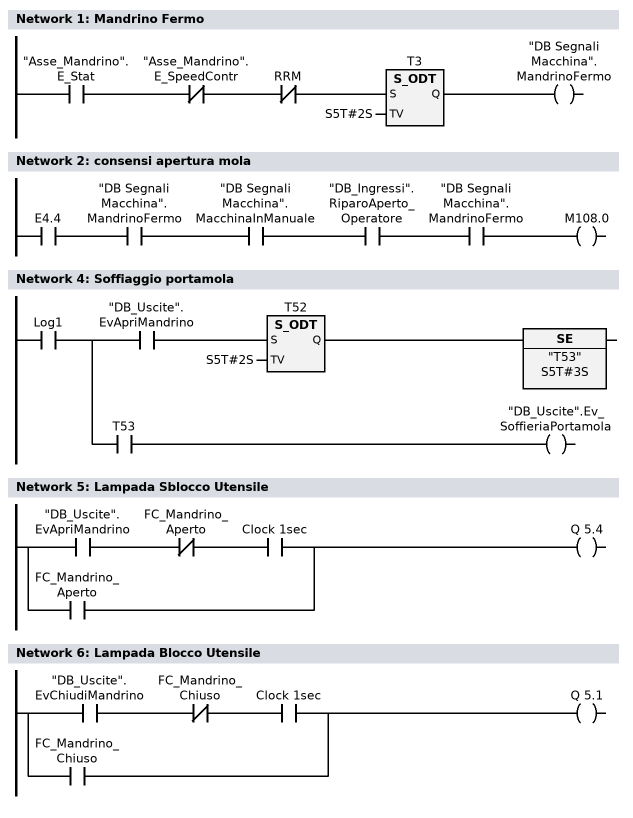
NETWORK
TITLE = Mandrino Fermo
      A     "Asse_Mandrino".E_Stat;
      AN    "Asse_Mandrino".E_SpeedContr;
      AN    "RRM";
      L     S5T#2S;
      SD    "T3";
      NOP   0;
      NOP   0;
      NOP   0;
      A     "T3";
      =     "DB Segnali Macchina".MandrinoFermo;
NETWORK
TITLE = consensi apertura mola
      A     "E4.4";
      A     "DB Segnali Macchina".MandrinoFermo;
      A     "DB Segnali Macchina".MacchinaInManuale;
      A     "DB_Ingressi".RiparoAperto_Operatore;
      A     "DB Segnali Macchina".MandrinoFermo;
      =     "M108.0";
NETWORK
TITLE = Blocco - Sblocco Mandrino
      A(;
      A(;
      A     "Pulsantiera.ChiudiMand";
      L     S5T#2S;
      SD    "T54";
      NOP   0;
      NOP   0;
      NOP   0;
      A     "T54";
      );
      A     "DB Segnali Macchina".MacchinaInManuale;
      A     "DB Segnali Macchina".MandrinoFermo;
      R     "DB_Uscite".EvApriMandrino;
      A(;
      A     "Pulsantiera.ApriMand";
      L     S5T#2S;
      SD    "T55";
      NOP   0;
      NOP   0;
      NOP   0;
      A     "T55";
      );
      A     "M108.0";
      S     "DB_Uscite".EvApriMandrino;
      A     "DB_Uscite".EvApriMandrino;
      );
      NOT;
      =     "DB_Uscite".EvChiudiMandrino;
NETWORK
TITLE = Soffiaggio portamola
      A     "Log1";
      =     L 0.0;
      A     L 0.0;
      A     "DB_Uscite".EvApriMandrino;
      L     S5T#2S;
      SD    "T52";
      NOP   0;
      NOP   0;
      NOP   0;
      A     "T52";
      L     S5T#3S;
      SE    "T53";
      A     L 0.0;
      A     "T53";
      =     "DB_Uscite".Ev_SoffieriaPortamola;
NETWORK
TITLE = Lampada Sblocco Utensile
      A     "DB_Uscite".EvApriMandrino;
      AN    "FC_Mandrino_Aperto";
      A     "Clock 1sec";
      O     "FC_Mandrino_Aperto";
      =     Q 5.4;
NETWORK
TITLE = Lampada Blocco Utensile
      A     "DB_Uscite".EvChiudiMandrino;
      AN    "FC_Mandrino_Chiuso";
      A     "Clock 1sec";
      O     "FC_Mandrino_Chiuso";
      =     Q 5.1;
END_FUNCTION

FUNCTION "FC Refrigerante" : VOID	// FC 106
TITLE = Gestione Refrigerante
AUTHOR : Asamec
VERSION : 0.1
BEGIN
NETWORK
TITLE = Refrigerante 1
      A(;
      A(;
      A     "Pulsantiera.AccendiOlio1";
      FP    "M10.0";
      =     "M93.2";
      A     "M93.2";
      AN    "DB_Ingressi".RiparoAperto_Operatore;
      A     "DB_Ingressi".RiparoChiuso_Robot;
      AN    "DB_Ingressi".Sel_MAN_AUTO;
      O     "M07";
      O;
      A     "M08";
      A(;
      L     "Chan1".T1;
      L     1;
      ==I;
      );
      );
      S     "M33.0";
      A(;
      O     "Pulsantiera.Reset";
      O;
      A     "Pulsantiera.SpegniOlio";
      AN    "DB_Ingressi".Sel_MAN_AUTO;
      ON    "DB Segnali Macchina".MacchinaAccesa;
      O     "M09";
      O;
      A     "M08";
      A(;
      L     "Chan1".T1;
      L     2;
      ==I;
      );
      A     "DB_Ingressi".Sel_MAN_AUTO;
      );
      R     "M33.0";
      A     "M33.0";
      );
      AN    "DB_Ingressi".RiparoAperto_Operatore;
      A     "DB_Ingressi".RiparoChiuso_Robot;
      AN    "M92.3";
      AN    "DB Allarmi".Canale1.Feed_And_Read_Disable.A510119;
      AN    "DB Allarmi".Canale1.Feed_And_Read_Disable.A510120;
      AN    "DB Allarmi".Canale1.Feed_Disable.A510004;
      AN    "DB Allarmi".Canale1.Feed_And_Read_Disable.A510117;
      =     "DB_Uscite".Olio1;
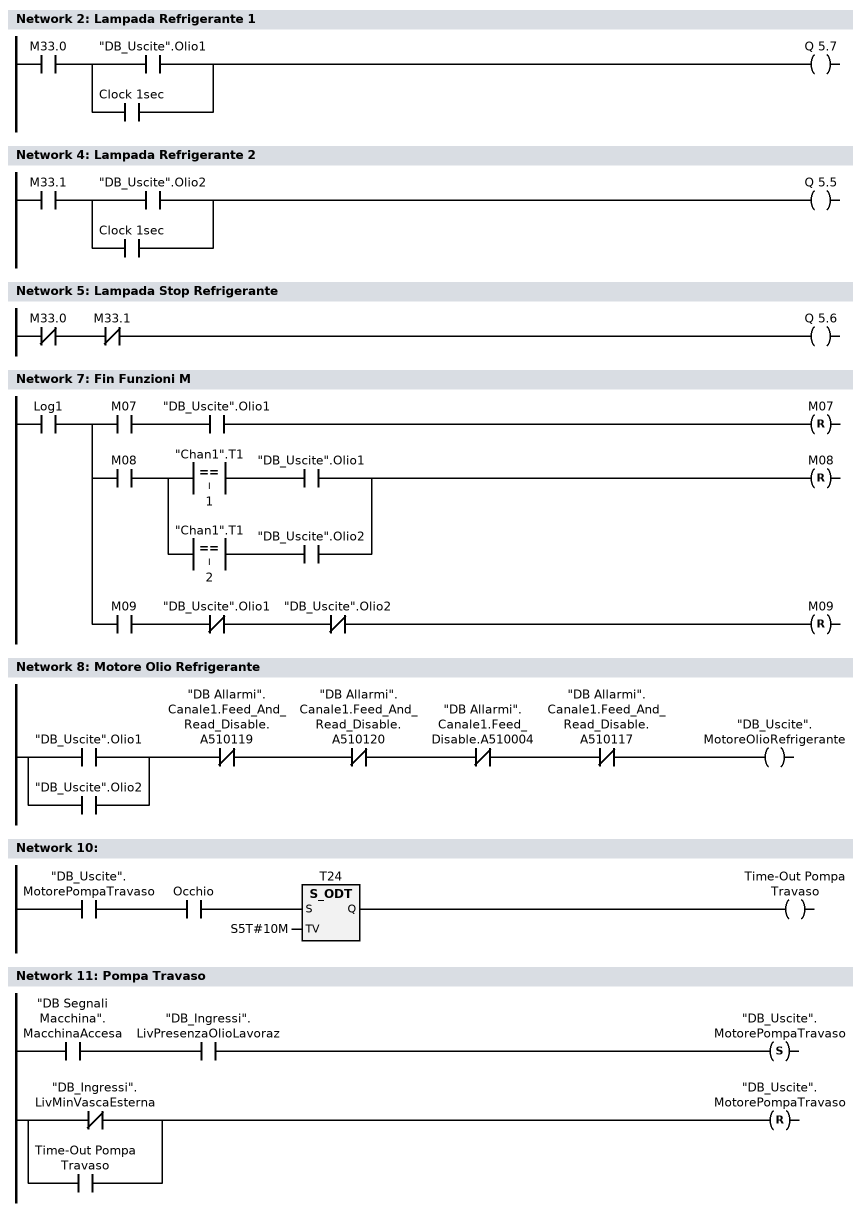
NETWORK
TITLE = Lampada Refrigerante 1
      A     "M33.0";
      A(;
      O     "DB_Uscite".Olio1;
      O     "Clock 1sec";
      );
      =     Q 5.7;
NETWORK
TITLE = Refrigerante 2
      A(;
      A(;
      A     "Pulsantiera.AccendiOlio2";
      FP    "M10.1";
      =     "M93.3";
      A     "M93.3";
      AN    "DB_Ingressi".RiparoAperto_Operatore;
      A     "DB_Ingressi".RiparoChiuso_Robot;
      AN    "DB_Ingressi".Sel_MAN_AUTO;
      O;
      A     "M08";
      A(;
      L     "Chan1".T1;
      L     2;
      ==I;
      );
      );
      S     "M33.1";
      A(;
      O     "Pulsantiera.Reset";
      O;
      A     "Pulsantiera.SpegniOlio";
      AN    "DB_Ingressi".Sel_MAN_AUTO;
      ON    "DB Segnali Macchina".MacchinaAccesa;
      O     "M09";
      O;
      A(;
      L     "Chan1".T1;
      L     1;
      ==I;
      );
      A     "DB_Ingressi".Sel_MAN_AUTO;
      );
      R     "M33.1";
      A     "M33.1";
      );
      AN    "DB_Ingressi".RiparoAperto_Operatore;
      A     "DB_Ingressi".RiparoChiuso_Robot;
      AN    "M92.3";
      AN    "DB Allarmi".Canale1.Feed_And_Read_Disable.A510119;
      AN    "DB Allarmi".Canale1.Feed_And_Read_Disable.A510120;
      AN    "DB Allarmi".Canale1.Feed_Disable.A510004;
      AN    "DB Allarmi".Canale1.Feed_And_Read_Disable.A510117;
      =     "DB_Uscite".Olio2;
NETWORK
TITLE = Lampada Refrigerante 2
      A     "M33.1";
      A(;
      O     "DB_Uscite".Olio2;
      O     "Clock 1sec";
      );
      =     Q 5.5;
NETWORK
TITLE = Lampada Stop Refrigerante
      AN    "M33.0";
      AN    "M33.1";
      =     Q 5.6;
NETWORK
TITLE = Sospendi refrigerante in automatico
      A     "Pulsantiera.SpegniOlio";
      A     "DB_Ingressi".Sel_MAN_AUTO;
      FP    "M93.1";
      X     "M92.3";
      =     "M92.3";
      A     "M07";
      O     "M08";
      ON    "DB_Ingressi".Sel_MAN_AUTO;
      R     "M92.3";
NETWORK
TITLE = Fin Funzioni M
      A     "Log1";
      =     L 0.0;
      A     L 0.0;
      A     "M07";
      A     "DB_Uscite".Olio1;
      R     "M07";
      A     L 0.0;
      A     "M08";
      A(;
      A(;
      L     "Chan1".T1;
      L     1;
      ==I;
      );
      A     "DB_Uscite".Olio1;
      O;
      A(;
      L     "Chan1".T1;
      L     2;
      ==I;
      );
      A     "DB_Uscite".Olio2;
      );
      R     "M08";
      A     L 0.0;
      A     "M09";
      AN    "DB_Uscite".Olio1;
      AN    "DB_Uscite".Olio2;
      R     "M09";
NETWORK
TITLE = Motore Olio Refrigerante
      A(;
      O     "DB_Uscite".Olio1;
      O     "DB_Uscite".Olio2;
      );
      AN    "DB Allarmi".Canale1.Feed_And_Read_Disable.A510119;
      AN    "DB Allarmi".Canale1.Feed_And_Read_Disable.A510120;
      AN    "DB Allarmi".Canale1.Feed_Disable.A510004;
      AN    "DB Allarmi".Canale1.Feed_And_Read_Disable.A510117;
      =     "DB_Uscite".MotoreOlioRefrigerante;
NETWORK
TITLE = Gestione Livelli
NETWORK
TITLE =
      A     "DB_Uscite".MotorePompaTravaso;
      A     "Occhio";
      L     S5T#10M;
      SD    "T24";
      NOP   0;
      NOP   0;
      NOP   0;
      A     "T24";
      =     "Time-Out Pompa Travaso";
NETWORK
TITLE = Pompa Travaso
      A     "DB Segnali Macchina".MacchinaAccesa;
      A     "DB_Ingressi".LivPresenzaOlioLavoraz;
      S     "DB_Uscite".MotorePompaTravaso;
      A(;
      ON    "DB_Ingressi".LivMinVascaEsterna;
      O     "Time-Out Pompa Travaso";
      );
      R     "DB_Uscite".MotorePompaTravaso;
      NOP   0;
NETWORK
TITLE =
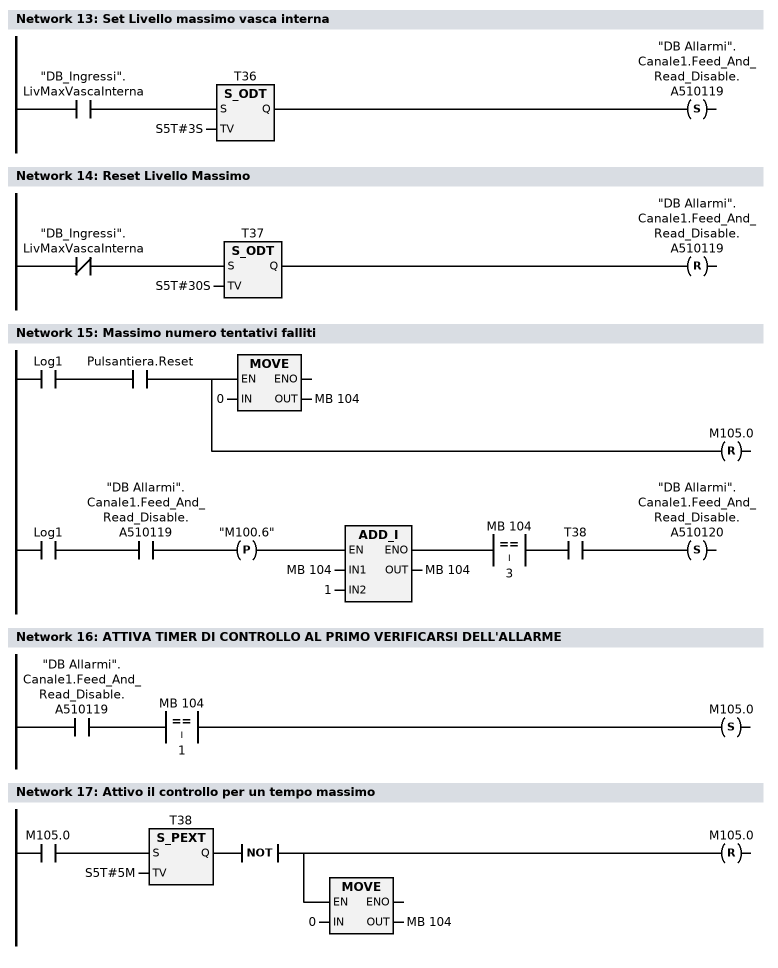
NETWORK
TITLE = Set Livello massimo vasca interna
      A     "DB_Ingressi".LivMaxVascaInterna;
      L     S5T#3S;
      SD    "T36";
      NOP   0;
      NOP   0;
      NOP   0;
      A     "T36";
      S     "DB Allarmi".Canale1.Feed_And_Read_Disable.A510119;
NETWORK
TITLE = Reset Livello Massimo
      AN    "DB_Ingressi".LivMaxVascaInterna;
      L     S5T#30S;
      SD    "T37";
      NOP   0;
      NOP   0;
      NOP   0;
      A     "T37";
      R     "DB Allarmi".Canale1.Feed_And_Read_Disable.A510119;
NETWORK
TITLE = Massimo numero tentativi falliti
      A     "Log1";
      =     L 0.0;
      A(;
      A     L 0.0;
      A     "DB Allarmi".Canale1.Feed_And_Read_Disable.A510119;
      FP    "M100.6";
      JNB   _001;
      L     MB 104;
      L     1;
      +I;
      T     MB 104;
      AN    OV;
      SAVE;
      CLR;
_001: A     BR;
      );
      A(;
      L     MB 104;
      L     3;
      ==I;
      );
      A     "T38";
      S     "DB Allarmi".Canale1.Feed_And_Read_Disable.A510120;
      A     L 0.0;
      A     "Pulsantiera.Reset";
      =     L 0.1;
      A     L 0.1;
      JNB   _002;
      L     0;
      T     MB 104;
_002: NOP   0;
      A     L 0.1;
      BLD   102;
      R     "M105.0";
NETWORK
TITLE = ATTIVA TIMER DI CONTROLLO AL PRIMO VERIFICARSI DELL'ALLARME
      A     "DB Allarmi".Canale1.Feed_And_Read_Disable.A510119;
      A(;
      L     MB 104;
      L     1;
      ==I;
      );
      S     "M105.0";
NETWORK
TITLE = Attivo il controllo per un tempo massimo
      A(;
      A     "M105.0";
      L     S5T#5M;
      SE    "T38";
      NOP   0;
      NOP   0;
      NOP   0;
      A     "T38";
      );
      NOT;
      =     L 0.0;
      A     L 0.0;
      BLD   102;
      R     "M105.0";
      A     L 0.0;
      JNB   _003;
      L     0;
      T     MB 104;
_003: NOP   0;
END_FUNCTION

FUNCTION "FC Assi" : VOID	// FC 107
VERSION : 0.1
BEGIN
NETWORK
TITLE =
NETWORK
TITLE = Abilita potenza OFF1 ( ex 48 - 112)
      A     "NC".E_DrivesInCylOp;
      A     "DB_Ingressi".AlimentatorePronto;
      A     "DB_Ingressi".PotenzaDriveInserita;
      S     "DB_Uscite".CdoOFF1;
      AN    "DB_Ingressi".PotenzaDriveInserita;
      R     "DB_Uscite".CdoOFF1;
NETWORK
TITLE = Abilita impulsi OFF3 ( ex 663 )
      A     "DB_Uscite".CdoOFF1;
      A     "DB_Ingressi".AusiliariInseriti;
//      U     "DB_Ingressi".PotenzaDriveInserita
      =     "DB_Uscite".CdoOFF3;
NETWORK
TITLE = Abilitazione assi
      A     "DB_Uscite".CdoOFF3;
//      U     "DB_Ingressi".ModuloARattivo
      =     "ConsensoRegolatore_X";
      =     "AbilitaImpulsi_X";
//-
      =     "ConsensoRegolatore_Y";
      =     "AbilitaImpulsi_Y";
//-
      =     "ConsensoRegolatore_Z";
      =     "AbilitaImpulsi_Z";
//-
NETWORK
TITLE = Abilitazione assi a e b (stop se fermi)
      A     "DB_Uscite".CdoOFF3;
      AN    "DB_Uscite".EV_ApriPortaPezzo;
      =     "M90.0";
      A     "Asse A in Direzione -";
      O     "Asse A in Direzione +";
      O     "BAG".E_AUTO;
      ON    "Chan1".E_ChanReset;
      A     "DB_Ingressi".AusiliariInseriti;
      S     "M90.1";
      R     "DB_Uscite".BloccoAsseA;
      A     "M90.0";
      A     "M90.1";
      AN    "DB_Ingressi".PressTavolaOrizzontale;
      AN    "DB_Uscite".EV_ApriPortaPezzo;
      L     S5T#200MS;
      SD    T 41;
//-
      A     T 41;
      S     "ConsensoRegolatore_A";
      S     "AbilitaImpulsi_A";
//-
      AN    "Asse A in Direzione -";
      AN    "Asse A in Direzione +";
      A     "Asse A Fermo";
      AN    "BAG".E_AUTO;
      A     "Chan1".E_ChanReset;
      L     S5T#40S;
      SD    T 42;
//-
      A     T 42;
      ON    "M90.0";
//      S     "DB_Uscite".BloccoAsseA
      R     "M90.1";
      A     T 42;
      ON    "M90.0";
      O     "DB_Uscite".EV_ApriPortaPezzo;
//      U     "DB_Uscite".BloccoAsseA
//      U     "DB_Ingressi".PressTavolaOrizzontale
      R     "ConsensoRegolatore_A";
      R     "AbilitaImpulsi_A";
NETWORK
TITLE = Abilita asse B
// per problemi legati al blocco - sblocco
// idraulico ho tolto i comandi
// per reinserirlo decommentare le righe
      A     "Asse B in Direzione -";
      O     "Asse B in Direzione +";
      O     "BAG".E_AUTO;
      ON    "Chan1".E_ChanReset;
      A     "DB_Ingressi".AusiliariInseriti;
      S     "M90.2";
      R     "DB_Uscite".BloccoAsseB;
      A     "M90.0";
      A     "M90.2";
      AN    "DB_Ingressi".PressTavolaVerticale;
      L     S5T#100MS;
      SD    T 43;
//-
      A     T 43;
      S     "ConsensoRegolatore_B";
      S     "AbilitaImpulsi_B";
//-
      AN    "Asse B in Direzione -";
      AN    "Asse B in Direzione +";
      A     "Asse B Fermo";
      AN    "BAG".E_AUTO;
      A     "Chan1".E_ChanReset;
      L     S5T#40S;
      SD    T 44;
//-
      A     T 44;
      ON    "M90.0";
//      S     "DB_Uscite".BloccoAsseB
      R     "M90.2";
//      U     "DB_Uscite".BloccoAsseB
//      U     "DB_Ingressi".PressTavolaVerticale
      R     "ConsensoRegolatore_B";
      R     "AbilitaImpulsi_B";
NETWORK
TITLE = Override
      L     IB 3;
      L     W#16#1F;
      AW;
      T     "Chan1".A_FD_OR;
      T     "Chan1".A_RT_OR;
      T     "Override Assi";
      SET;
      S     "Chan1".A_RT_ORA;
      S     "Chan1".A_FD_ORA;
NETWORK
TITLE = Feed Stop
      A     "Pulsantiera.FeedHold";
      O     "Pulsatiera.SpindleHold";
      O     "DB Segnali Macchina".BloccoAssiAttivo;
      O     "DB Segnali Macchina".BloccoMandrinoAttivo;
      O     "DB Segnali Macchina".BloccoAssiEMandrinoAttiv;
      =     "Feed Stop";
NETWORK
TITLE = Spindle Stop
      A     "Pulsatiera.SpindleHold";
      ON    "DB_Uscite".EvChiudiMandrino;
      ON    "FC_Mandrino_Chiuso";
      O     "DB Segnali Macchina".BloccoMandrinoAttivo;
      O     "DB Segnali Macchina".BloccoAssiEMandrinoAttiv;
      =     "SpindleStop";
NETWORK
TITLE = comandi al mandrino
      L     "Asse_Mandrino".E_MFunct;
      L     0;
      ==I;
      JC    M111;
//-
      L     "Asse_Mandrino".E_MFunct;
      L     3;
      ==I;
      S     "RRM";
//-
      L     "Asse_Mandrino".E_MFunct;
      L     4;
      ==I;
      S     "RRM";
//-
      L     "Asse_Mandrino".E_MFunct;
      L     5;
      ==I;
      R     "RRM";
//-
      L     0;
      T     "Asse_Mandrino".E_MFunct;
M111: NOP   0;
      A     "Chan1".A_Reset;
      R     "RRM";
      A     "M03";
      O     "M04";
      A     "RRM";
      A     "Asse_Mandrino".E_SpeedContr;
      A     "Asse_Mandrino".E_NactNset;
      AN    "Mandrino Fermo";
      R     "M03";
      R     "M04";
      A     "M05";
      AN    "RRM";
      A     "Mandrino Fermo";
      R     "M05";
      A     "RRM";
      S     "AbilitaImpulsi_Mandrino";
      S     "ConsensoRegolatore_Mandr";
      AN    "RRM";
      A     "Mandrino Fermo";
      R     "AbilitaImpulsi_Mandrino";
      R     "ConsensoRegolatore_Mandr";
NETWORK
TITLE = comandi al mandrino diamantatura
//-  comando di giri
      L     "Chan1".H1;
      L     1.600000e+02;
      /R;
      T     "MD171";
//- mandrino a regime
      L     "MD171";
      L     "MD176";
      -R;
      T     "MD180";
      L     "MD180";
      ABS;
      L     1.000000e+01;
      <R;
      =     "M175.5";
//- mandrino fermo
      L     "MD176";
      ABS;
      L     1.000000e+00;
      <R;
      =     "M175.6";
//- comando di rotazione
      A     "M13";
      S     "RRM2";
      R     "M170.1";
//-
      A     "M14";
      S     "RRM2";
      S     "M170.1";
//-
      A     "M13";
      O     "M14";
      A     "M175.5";
      L     S5T#1S;
      SD    "T21";
//-
      A     "T21";
      R     "M13";
      R     "M14";
//-
      A     "M15";
      O     "Chan1".A_Reset;
      R     "RRM2";
      AN    "RRM2";
      A     "M175.6";
      R     "M15";
//-
      A     "M13";
      O     "M14";
      L     S5T#500MS;
      SP    "T22";
//-
      A     "RRM2";
      AN    "T22";
      AN    "SpindleStop";
      =     "M170.0";
      A     "M175.1";
      O     "M175.2";
      A     "Chan1".A_Reset;
      =     "M170.2";
NETWORK
TITLE = comando freni assi - Y
      A     "DB Segnali Macchina".MacchinaAccesaRitardato;
// U asse in coppia
      =     "DB_Uscite".SbloccoFrenoAsseY;
NETWORK
TITLE = Gestione Asse X
      CALL  "FC Intrefaccia Assi" (
           OVERR_ACT                := TRUE,
           FUNZ_PUNT                := FALSE,
           RIC_FUNZ_PUNT            := FALSE,
           CONS_REGOL               := "ConsensoRegolatore_X",
           ABIL_IMP                 := "AbilitaImpulsi_X",
           ATT_CAM_SW               := FALSE,
           FC_SOFTWARE2_PIU         := FALSE,
           FC_SOFTWARE2_MENO        := FALSE,
           CONS_AVANZ               := "Feed Stop",
           OLTREC_PIU               := FALSE,
           CANC_PERC_RES            := FALSE,
           BLOC_AX                  := FALSE,
           LIMIT_VEL                := FALSE,
           OVERR_RAP_ACT            := TRUE,
           JOG_STANDARD             := TRUE,
           JOG_MENO                 := FALSE,
           JOG_PIU                  := FALSE,
           VAL_INCR                 := B#16#0,
           OLTREC_MENO              := FALSE,
           VAL_OVERR                := "Override Assi",
           DB_INT_AX                := 31,
           SIST_MIS_1               := TRUE,
           SIST_MIS_2               := FALSE,
           AX_CAMME_REF             := FALSE,
           PUNTO_REF_1              := FALSE,
           MOV_AX                   := "Asse X in Movimento",
           MOV_AX_MENO              := "Asse X in Direzione -",
           MOV_AX_PIU               := "Asse X in Direzione +",
           ASSE_FERMO               := "Asse X Fermo",
           ASSE_AZZER               := "Asse X Azzerato");
NETWORK
TITLE = Gestione Asse Y
      CALL  "FC Intrefaccia Assi" (
           OVERR_ACT                := TRUE,
           FUNZ_PUNT                := FALSE,
           RIC_FUNZ_PUNT            := FALSE,
           CONS_REGOL               := "ConsensoRegolatore_Y",
           ABIL_IMP                 := "AbilitaImpulsi_Y",
           ATT_CAM_SW               := FALSE,
           FC_SOFTWARE2_PIU         := FALSE,
           FC_SOFTWARE2_MENO        := FALSE,
           CONS_AVANZ               := "Feed Stop",
           OLTREC_PIU               := FALSE,
           CANC_PERC_RES            := FALSE,
           BLOC_AX                  := FALSE,
           LIMIT_VEL                := FALSE,
           OVERR_RAP_ACT            := TRUE,
           JOG_STANDARD             := TRUE,
           JOG_MENO                 := FALSE,
           JOG_PIU                  := FALSE,
           VAL_INCR                 := B#16#0,
           OLTREC_MENO              := FALSE,
           VAL_OVERR                := "Override Assi",
           DB_INT_AX                := 32,
           SIST_MIS_1               := TRUE,
           SIST_MIS_2               := FALSE,
           AX_CAMME_REF             := FALSE,
           PUNTO_REF_1              := FALSE,
           MOV_AX                   := "Asse Y in Movimento",
           MOV_AX_MENO              := "Asse Y in Direzione -",
           MOV_AX_PIU               := "Asse Y in Direzione +",
           ASSE_FERMO               := "Asse Y Fermo",
           ASSE_AZZER               := "Asse Y Azzerato");
NETWORK
TITLE = Gestione Asse Z
      CALL  "FC Intrefaccia Assi" (
           OVERR_ACT                := TRUE,
           FUNZ_PUNT                := FALSE,
           RIC_FUNZ_PUNT            := FALSE,
           CONS_REGOL               := "ConsensoRegolatore_Z",
           ABIL_IMP                 := "AbilitaImpulsi_Z",
           ATT_CAM_SW               := FALSE,
           FC_SOFTWARE2_PIU         := FALSE,
           FC_SOFTWARE2_MENO        := FALSE,
           CONS_AVANZ               := "Feed Stop",
           OLTREC_PIU               := FALSE,
           CANC_PERC_RES            := FALSE,
           BLOC_AX                  := FALSE,
           LIMIT_VEL                := FALSE,
           OVERR_RAP_ACT            := TRUE,
           JOG_STANDARD             := TRUE,
           JOG_MENO                 := FALSE,
           JOG_PIU                  := FALSE,
           VAL_INCR                 := B#16#0,
           OLTREC_MENO              := FALSE,
           VAL_OVERR                := "Override Assi",
           DB_INT_AX                := 33,
           SIST_MIS_1               := TRUE,
           SIST_MIS_2               := FALSE,
           AX_CAMME_REF             := FALSE,
           PUNTO_REF_1              := FALSE,
           MOV_AX                   := "Asse Z in Movimento",
           MOV_AX_MENO              := "Asse Z in Direzione -",
           MOV_AX_PIU               := "Asse Z in Direzione +",
           ASSE_FERMO               := "Asse Z Fermo",
           ASSE_AZZER               := "Asse Z Azzerato");
NETWORK
TITLE = Gestione Asse A
      CALL  "FC Intrefaccia Assi" (
           OVERR_ACT                := TRUE,
           FUNZ_PUNT                := FALSE,
           RIC_FUNZ_PUNT            := FALSE,
           CONS_REGOL               := "ConsensoRegolatore_A",
           ABIL_IMP                 := "AbilitaImpulsi_A",
           ATT_CAM_SW               := FALSE,
           FC_SOFTWARE2_PIU         := FALSE,
           FC_SOFTWARE2_MENO        := FALSE,
           CONS_AVANZ               := "Feed Stop",
           OLTREC_PIU               := FALSE,
           CANC_PERC_RES            := FALSE,
           BLOC_AX                  := FALSE,
           LIMIT_VEL                := FALSE,
           OVERR_RAP_ACT            := TRUE,
           JOG_STANDARD             := TRUE,
           JOG_MENO                 := FALSE,
           JOG_PIU                  := FALSE,
           VAL_INCR                 := B#16#0,
           OLTREC_MENO              := FALSE,
           VAL_OVERR                := "Override Assi",
           DB_INT_AX                := 34,
           SIST_MIS_1               := TRUE,
           SIST_MIS_2               := FALSE,
           AX_CAMME_REF             := FALSE,
           PUNTO_REF_1              := FALSE,
           MOV_AX                   := "Asse A in Movimento",
           MOV_AX_MENO              := "Asse A in Direzione -",
           MOV_AX_PIU               := "Asse A in Direzione +",
           ASSE_FERMO               := "Asse A Fermo",
           ASSE_AZZER               := "Asse A Azzerato");
NETWORK
TITLE = Gestione Asse B
      CALL  "FC Intrefaccia Assi" (
           OVERR_ACT                := TRUE,
           FUNZ_PUNT                := FALSE,
           RIC_FUNZ_PUNT            := FALSE,
           CONS_REGOL               := "ConsensoRegolatore_B",
           ABIL_IMP                 := "AbilitaImpulsi_B",
           ATT_CAM_SW               := FALSE,
           FC_SOFTWARE2_PIU         := FALSE,
           FC_SOFTWARE2_MENO        := FALSE,
           CONS_AVANZ               := "Feed Stop",
           OLTREC_PIU               := FALSE,
           CANC_PERC_RES            := FALSE,
           BLOC_AX                  := FALSE,
           LIMIT_VEL                := FALSE,
           OVERR_RAP_ACT            := TRUE,
           JOG_STANDARD             := TRUE,
           JOG_MENO                 := FALSE,
           JOG_PIU                  := FALSE,
           VAL_INCR                 := B#16#0,
           OLTREC_MENO              := FALSE,
           VAL_OVERR                := "Override Assi",
           DB_INT_AX                := 35,
           SIST_MIS_1               := TRUE,
           SIST_MIS_2               := FALSE,
           AX_CAMME_REF             := FALSE,
           PUNTO_REF_1              := FALSE,
           MOV_AX                   := "Asse B in Movimento",
           MOV_AX_MENO              := "Asse B in Direzione -",
           MOV_AX_PIU               := "Asse B in Direzione +",
           ASSE_FERMO               := "Asse B Fermo",
           ASSE_AZZER               := "Asse B Azzerato");
NETWORK
TITLE = Gestione Mandrino
      CALL  "FC Intrefaccia Assi" (
           OVERR_ACT                := TRUE,
           FUNZ_PUNT                := FALSE,
           RIC_FUNZ_PUNT            := FALSE,
           CONS_REGOL               := "ConsensoRegolatore_Mandr",
           ABIL_IMP                 := "AbilitaImpulsi_Mandrino",
           ATT_CAM_SW               := FALSE,
           FC_SOFTWARE2_PIU         := FALSE,
           FC_SOFTWARE2_MENO        := FALSE,
           CONS_AVANZ               := "SpindleStop",
           OLTREC_PIU               := FALSE,
           CANC_PERC_RES            := FALSE,
           BLOC_AX                  := FALSE,
           LIMIT_VEL                := FALSE,
           OVERR_RAP_ACT            := TRUE,
           JOG_STANDARD             := TRUE,
           JOG_MENO                 := FALSE,
           JOG_PIU                  := FALSE,
           VAL_INCR                 := B#16#0,
           OLTREC_MENO              := FALSE,
           VAL_OVERR                := "Override Assi",
           DB_INT_AX                := 36,
           SIST_MIS_1               := TRUE,
           SIST_MIS_2               := FALSE,
           AX_CAMME_REF             := FALSE,
           PUNTO_REF_1              := FALSE,
           MOV_AX                   := "Mandrino in Movimento",
           MOV_AX_MENO              := "Mandrino in Direzione -",
           MOV_AX_PIU               := "Mandrino in Direzione +",
           ASSE_FERMO               := "Mandrino Fermo",
           ASSE_AZZER               := "Mandrino Azzerato");
NETWORK
TITLE = Mandrino di diamantatura
      CALL  "FC_Profibus_MM4" (
           Periferic_Address        := 288,
           Drive_On_Off             := "M170.0",
           Drive_Reversing          := "M170.1",
           Drive_Fault_ACKN         := "M170.2",
           Drive_F_Setpoint         := "MD171",
           Drive_in_operation       := "M175.0",
           Drive_Fault_Active       := "M175.1",
           Drive_Alarm_Active       := "M175.2",
           Freno                    := M 175.3,
           Drive_F_Act              := "MD176");
END_FUNCTION

FUNCTION "FC Lubrificazioni" : VOID	// FC 108
VERSION : 0.1
VAR_TEMP
  TempoLub : S5TIME ;
  Intervallo : S5TIME ;
  AppTempo : INT ;
  AppTempo2 : S5TIME ;
END_VAR
BEGIN
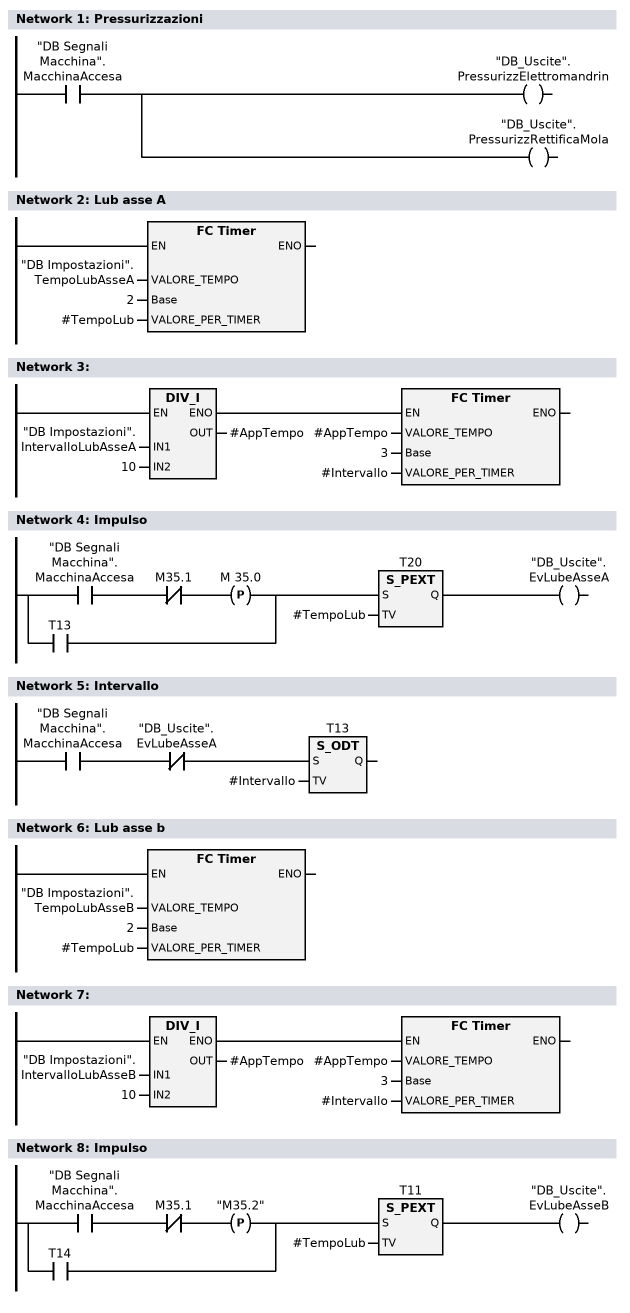
NETWORK
TITLE = Pressurizzazioni
      A     "DB Segnali Macchina".MacchinaAccesa;
      =     "DB_Uscite".PressurizzElettromandrin;
      =     "DB_Uscite".PressurizzRettificaMola;
NETWORK
TITLE = Lub asse A
      CALL  "FC Timer" (
           VALORE_TEMPO             := "DB Impostazioni".TempoLubAsseA,
           Base                     := 2,
           VALORE_PER_TIMER         := #TempoLub);
      NOP   0;
NETWORK
TITLE =
      A(;
      L     "DB Impostazioni".IntervalloLubAsseA;
      L     10;
      /I;
      T     #AppTempo;
      AN    OV;
      SAVE;
      CLR;
      A     BR;
      );
      JNB   _001;
      CALL  "FC Timer" (
           VALORE_TEMPO             := #AppTempo,
           Base                     := 3,
           VALORE_PER_TIMER         := #Intervallo);
_001: NOP   0;
NETWORK
TITLE = Impulso
      A(;
      A     "DB Segnali Macchina".MacchinaAccesa;
      AN    "M35.1";
      FP    M 35.0;
      O     "T13";
      );
      L     #TempoLub;
      SE    "T20";
      NOP   0;
      NOP   0;
      NOP   0;
      A     "T20";
      =     "DB_Uscite".EvLubeAsseA;
NETWORK
TITLE = Intervallo
      A     "DB Segnali Macchina".MacchinaAccesa;
      AN    "DB_Uscite".EvLubeAsseA;
      L     #Intervallo;
      SD    "T13";
      NOP   0;
      NOP   0;
      NOP   0;
      NOP   0;
NETWORK
TITLE = Lub asse b
      CALL  "FC Timer" (
           VALORE_TEMPO             := "DB Impostazioni".TempoLubAsseB,
           Base                     := 2,
           VALORE_PER_TIMER         := #TempoLub);
      NOP   0;
NETWORK
TITLE =
      A(;
      L     "DB Impostazioni".IntervalloLubAsseB;
      L     10;
      /I;
      T     #AppTempo;
      AN    OV;
      SAVE;
      CLR;
      A     BR;
      );
      JNB   _002;
      CALL  "FC Timer" (
           VALORE_TEMPO             := #AppTempo,
           Base                     := 3,
           VALORE_PER_TIMER         := #Intervallo);
_002: NOP   0;
NETWORK
TITLE = Impulso
      A(;
      A     "DB Segnali Macchina".MacchinaAccesa;
      AN    "M35.1";
      FP    "M35.2";
      O     "T14";
      );
      L     #TempoLub;
      SE    "T11";
      NOP   0;
      NOP   0;
      NOP   0;
      A     "T11";
      =     "DB_Uscite".EvLubeAsseB;
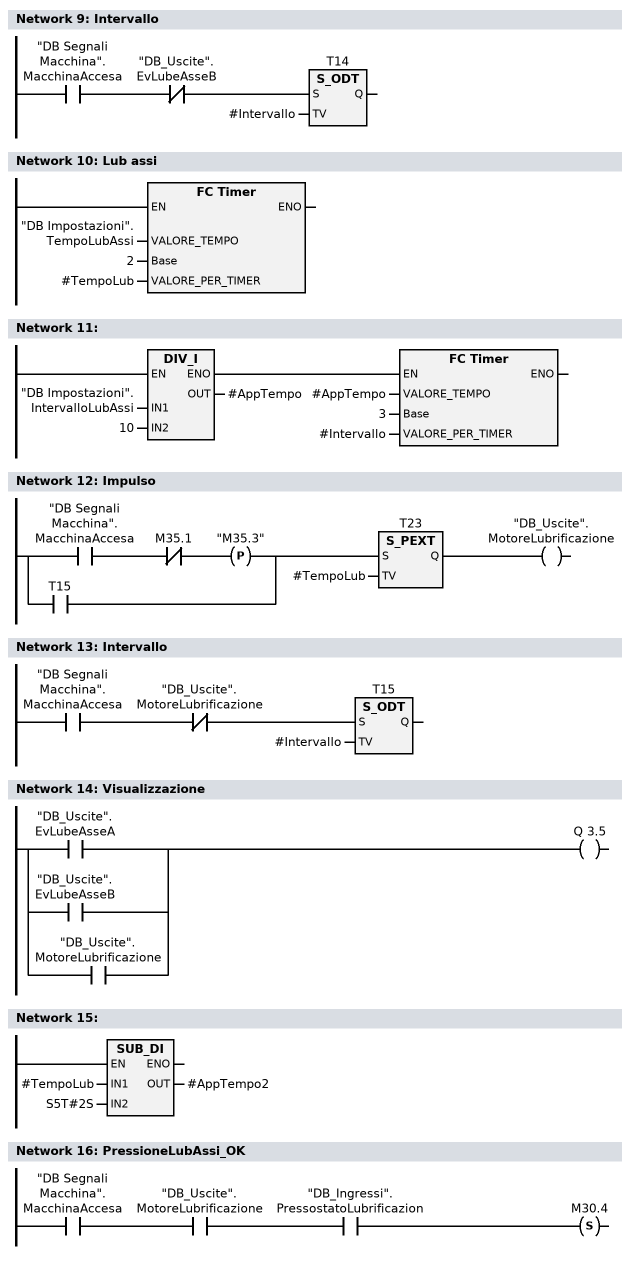
NETWORK
TITLE = Intervallo
      A     "DB Segnali Macchina".MacchinaAccesa;
      AN    "DB_Uscite".EvLubeAsseB;
      L     #Intervallo;
      SD    "T14";
      NOP   0;
      NOP   0;
      NOP   0;
      NOP   0;
NETWORK
TITLE = Lub assi
      CALL  "FC Timer" (
           VALORE_TEMPO             := "DB Impostazioni".TempoLubAssi,
           Base                     := 2,
           VALORE_PER_TIMER         := #TempoLub);
      NOP   0;
NETWORK
TITLE =
      A(;
      L     "DB Impostazioni".IntervalloLubAssi;
      L     10;
      /I;
      T     #AppTempo;
      AN    OV;
      SAVE;
      CLR;
      A     BR;
      );
      JNB   _003;
      CALL  "FC Timer" (
           VALORE_TEMPO             := #AppTempo,
           Base                     := 3,
           VALORE_PER_TIMER         := #Intervallo);
_003: NOP   0;
NETWORK
TITLE = Impulso
      A(;
      A     "DB Segnali Macchina".MacchinaAccesa;
      AN    "M35.1";
      FP    "M35.3";
      O     "T15";
      );
      L     #TempoLub;
      SE    "T23";
      NOP   0;
      NOP   0;
      NOP   0;
      A     "T23";
      =     "DB_Uscite".MotoreLubrificazione;
NETWORK
TITLE = Intervallo
      A     "DB Segnali Macchina".MacchinaAccesa;
      AN    "DB_Uscite".MotoreLubrificazione;
      L     #Intervallo;
      SD    "T15";
      NOP   0;
      NOP   0;
      NOP   0;
      NOP   0;
NETWORK
TITLE = Visualizzazione
      O     "DB_Uscite".EvLubeAsseA;
      O     "DB_Uscite".EvLubeAsseB;
      O     "DB_Uscite".MotoreLubrificazione;
      =     Q 3.5;
NETWORK
TITLE =
      L     #TempoLub;
      L     S5T#2S;
      -D;
      T     #AppTempo2;
NETWORK
TITLE = PressioneLubAssi_OK
      A     "DB Segnali Macchina".MacchinaAccesa;
      A     "DB_Uscite".MotoreLubrificazione;
      A     "DB_Ingressi".PressostatoLubrificazion;
      S     "M30.4";
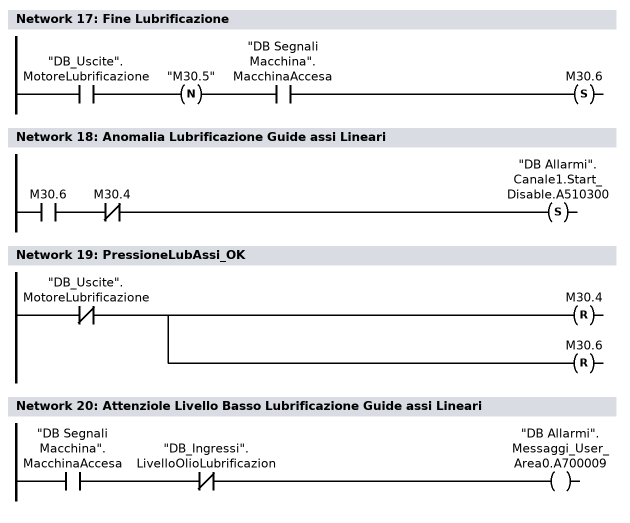
NETWORK
TITLE = Fine Lubrificazione
      A     "DB_Uscite".MotoreLubrificazione;
      FN    "M30.5";
      A     "DB Segnali Macchina".MacchinaAccesa;
      S     "M30.6";
NETWORK
TITLE = Anomalia Lubrificazione Guide assi Lineari
      A     "M30.6";
      AN    "M30.4";
      S     "DB Allarmi".Canale1.Start_Disable.A510300;
NETWORK
TITLE = PressioneLubAssi_OK
      AN    "DB_Uscite".MotoreLubrificazione;
      R     "M30.4";
      R     "M30.6";
NETWORK
TITLE = Attenziole Livello Basso Lubrificazione Guide assi Lineari
      A     "DB Segnali Macchina".MacchinaAccesa;
      AN    "DB_Ingressi".LivelloOlioLubrificazion;
      =     "DB Allarmi".Messaggi_User_Area0.A700009;
END_FUNCTION

FUNCTION "FC Idraulica" : VOID	// FC 110
VERSION : 0.1
BEGIN
NETWORK
TITLE = GEstione elementi idraulici generali
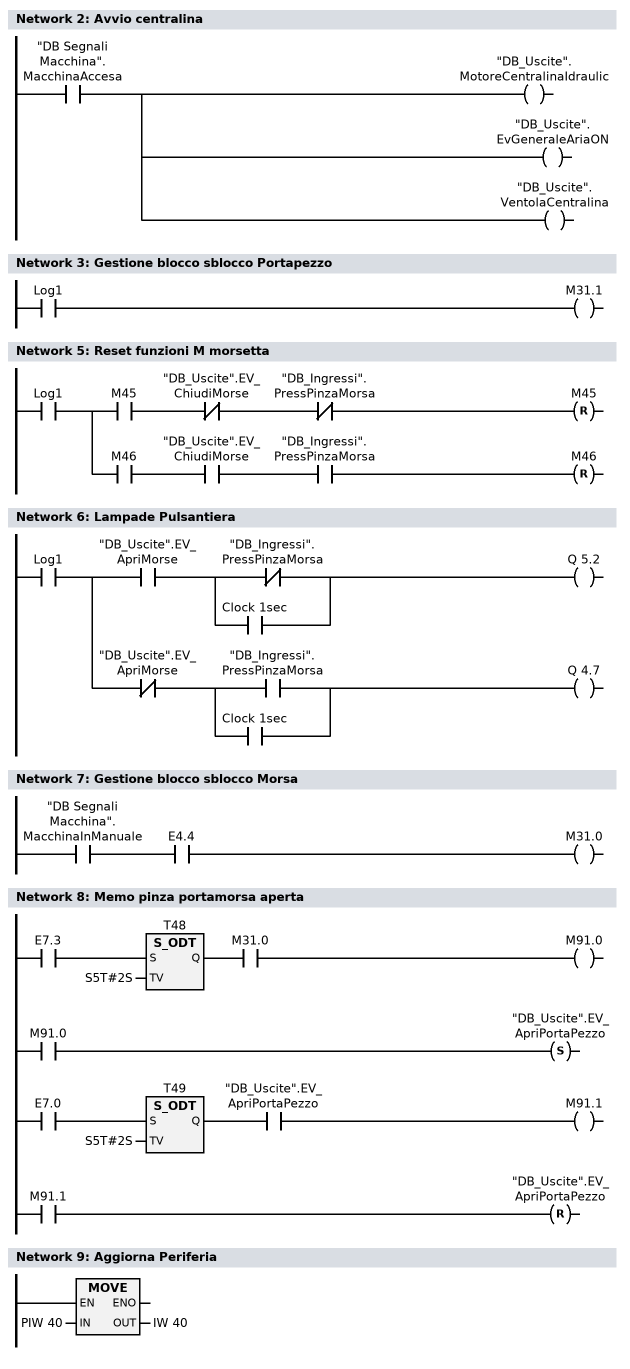
NETWORK
TITLE = Avvio centralina
      A     "DB Segnali Macchina".MacchinaAccesa;
      =     "DB_Uscite".MotoreCentralinaIdraulic;
      =     "DB_Uscite".EvGeneraleAriaON;
      =     "DB_Uscite".VentolaCentralina;
NETWORK
TITLE = Gestione blocco sblocco Portapezzo
      A     "Log1";
      =     "M31.1";
NETWORK
TITLE = Memo pinza morsa portapezzo
      A(;
      A(;
      A(;
      A     "E7.2";
      L     S5T#2S;
      SD    "T46";
      NOP   0;
      NOP   0;
      NOP   0;
      A     "T46";
      );
      A     "M31.1";
      O;
      A     "M45";
      A     "M31.1";
      O     "M51.2";
      );
      S     "DB_Uscite".EV_ApriMorse;
      A(;
      A(;
      A     "E6.7";
      L     S5T#2S;
      SD    "T47";
      NOP   0;
      NOP   0;
      NOP   0;
      A     "T47";
      );
      A     "M31.1";
      O;
      A     "M46";
      A     "M31.1";
      O     "M51.3";
      );
      R     "DB_Uscite".EV_ApriMorse;
      A     "DB_Uscite".EV_ApriMorse;
      );
      NOT;
      =     "DB_Uscite".EV_ChiudiMorse;
NETWORK
TITLE = Reset funzioni M morsetta
      A     "Log1";
      =     L 0.0;
      A     L 0.0;
      A     "M45";
      AN    "DB_Uscite".EV_ChiudiMorse;
      AN    "DB_Ingressi".PressPinzaMorsa;
      R     "M45";
      A     L 0.0;
      A     "M46";
      A     "DB_Uscite".EV_ChiudiMorse;
      A     "DB_Ingressi".PressPinzaMorsa;
      R     "M46";
NETWORK
TITLE = Lampade Pulsantiera
      A     "Log1";
      =     L 0.0;
      A     L 0.0;
      A     "DB_Uscite".EV_ApriMorse;
      A(;
      ON    "DB_Ingressi".PressPinzaMorsa;
      O     "Clock 1sec";
      );
      =     Q 5.2;
      A     L 0.0;
      AN    "DB_Uscite".EV_ApriMorse;
      A(;
      O     "DB_Ingressi".PressPinzaMorsa;
      O     "Clock 1sec";
      );
      =     Q 4.7;
NETWORK
TITLE = Gestione blocco sblocco Morsa
      A     "DB Segnali Macchina".MacchinaInManuale;
      A     "E4.4";
      =     "M31.0";
NETWORK
TITLE = Memo pinza portamorsa aperta
      A(;
      A     "E7.3";
      L     S5T#2S;
      SD    "T48";
      NOP   0;
      NOP   0;
      NOP   0;
      A     "T48";
      );
      A     "M31.0";
      =     "M91.0";
      A     "M91.0";
      S     "DB_Uscite".EV_ApriPortaPezzo;
      A(;
      A     "E7.0";
      L     S5T#2S;
      SD    "T49";
      NOP   0;
      NOP   0;
      NOP   0;
      A     "T49";
      );
      A     "DB_Uscite".EV_ApriPortaPezzo;
      =     "M91.1";
      A     "M91.1";
      R     "DB_Uscite".EV_ApriPortaPezzo;
      NOP   0;
NETWORK
TITLE = Aggiorna Periferia
      L     PIW 40;
      T     IW 40;
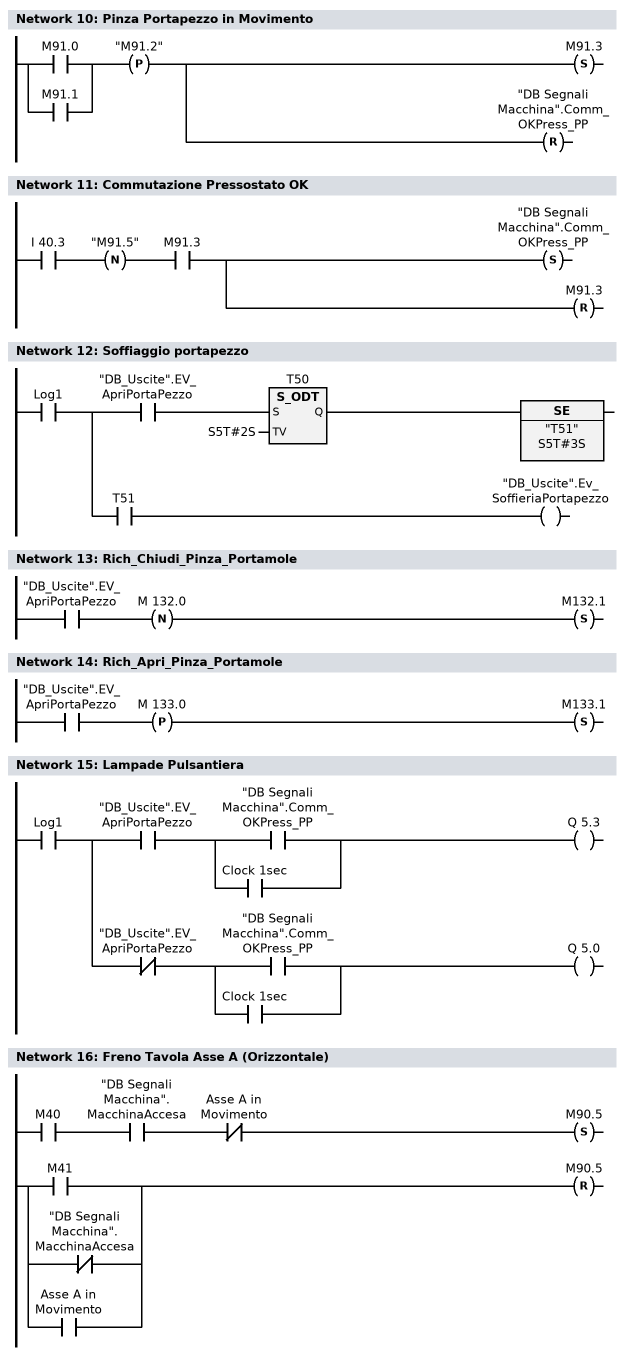
NETWORK
TITLE = Pinza Portapezzo in Movimento
      A(;
      O     "M91.0";
      O     "M91.1";
      );
      FP    "M91.2";
      S     "M91.3";
      R     "DB Segnali Macchina".Comm_OKPress_PP;
NETWORK
TITLE = Commutazione Pressostato OK
      A     I 40.3;
      FN    "M91.5";
      A     "M91.3";
      S     "DB Segnali Macchina".Comm_OKPress_PP;
      R     "M91.3";
NETWORK
TITLE = Soffiaggio portapezzo
      A     "Log1";
      =     L 0.0;
      A     L 0.0;
      A     "DB_Uscite".EV_ApriPortaPezzo;
      L     S5T#2S;
      SD    "T50";
      NOP   0;
      NOP   0;
      NOP   0;
      A     "T50";
      L     S5T#3S;
      SE    "T51";
      A     L 0.0;
      A     "T51";
      =     "DB_Uscite".Ev_SoffieriaPortapezzo;
NETWORK
TITLE = Rich_Chiudi_Pinza_Portamole
      A     "DB_Uscite".EV_ApriPortaPezzo;
      FN    M 132.0;
      S     "M132.1";
NETWORK
TITLE = Rich_Apri_Pinza_Portamole
      A     "DB_Uscite".EV_ApriPortaPezzo;
      FP    M 133.0;
      S     "M133.1";
NETWORK
TITLE = Lampade Pulsantiera
      A     "Log1";
      =     L 0.0;
      A     L 0.0;
      A     "DB_Uscite".EV_ApriPortaPezzo;
      A(;
      O     "DB Segnali Macchina".Comm_OKPress_PP;
      O     "Clock 1sec";
      );
      =     Q 5.3;
      A     L 0.0;
      AN    "DB_Uscite".EV_ApriPortaPezzo;
      A(;
      O     "DB Segnali Macchina".Comm_OKPress_PP;
      O     "Clock 1sec";
      );
      =     Q 5.0;
NETWORK
TITLE = Freno Tavola Asse A (Orizzontale)
      A     "M40";
      A     "DB Segnali Macchina".MacchinaAccesa;
      AN    "Asse A in Movimento";
      S     "M90.5";
      A(;
      O     "M41";
      ON    "DB Segnali Macchina".MacchinaAccesa;
      O     "Asse A in Movimento";
      );
      R     "M90.5";
      NOP   0;
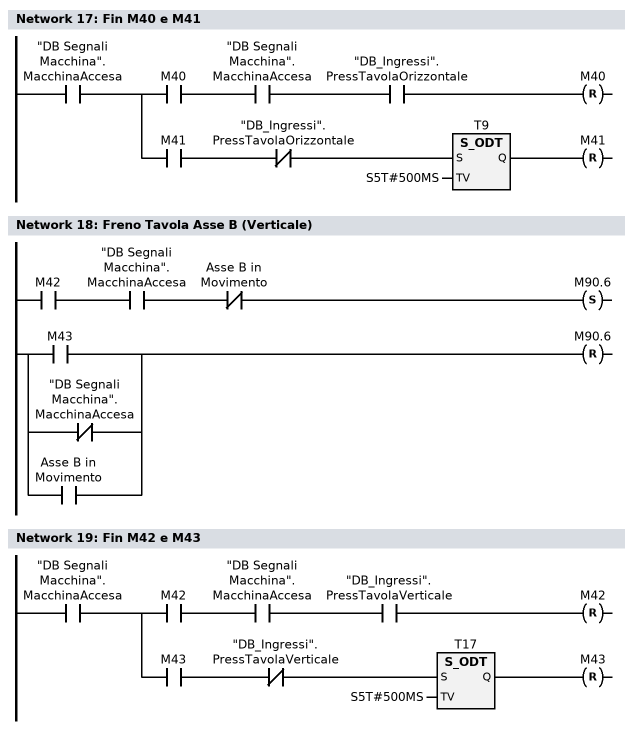
NETWORK
TITLE = Fin M40 e M41
      A     "DB Segnali Macchina".MacchinaAccesa;
      =     L 0.0;
      A     L 0.0;
      A     "M40";
      A     "DB Segnali Macchina".MacchinaAccesa;
      A     "DB_Ingressi".PressTavolaOrizzontale;
      R     "M40";
      A     L 0.0;
      A     "M41";
      AN    "DB_Ingressi".PressTavolaOrizzontale;
      L     S5T#500MS;
      SD    "T9";
      NOP   0;
      NOP   0;
      NOP   0;
      A     "T9";
      R     "M41";
NETWORK
TITLE = Freno Tavola Asse B (Verticale)
      A     "M42";
      A     "DB Segnali Macchina".MacchinaAccesa;
      AN    "Asse B in Movimento";
      S     "M90.6";
      A(;
      O     "M43";
      ON    "DB Segnali Macchina".MacchinaAccesa;
      O     "Asse B in Movimento";
      );
      R     "M90.6";
      NOP   0;
NETWORK
TITLE = Fin M42 e M43
      A     "DB Segnali Macchina".MacchinaAccesa;
      =     L 0.0;
      A     L 0.0;
      A     "M42";
      A     "DB Segnali Macchina".MacchinaAccesa;
      A     "DB_Ingressi".PressTavolaVerticale;
      R     "M42";
      A     L 0.0;
      A     "M43";
      AN    "DB_Ingressi".PressTavolaVerticale;
      L     S5T#500MS;
      SD    "T17";
      NOP   0;
      NOP   0;
      NOP   0;
      A     "T17";
      R     "M43";
END_FUNCTION

FUNCTION "FC Ausiliari" : VOID	// FC 111
VERSION : 0.1
BEGIN
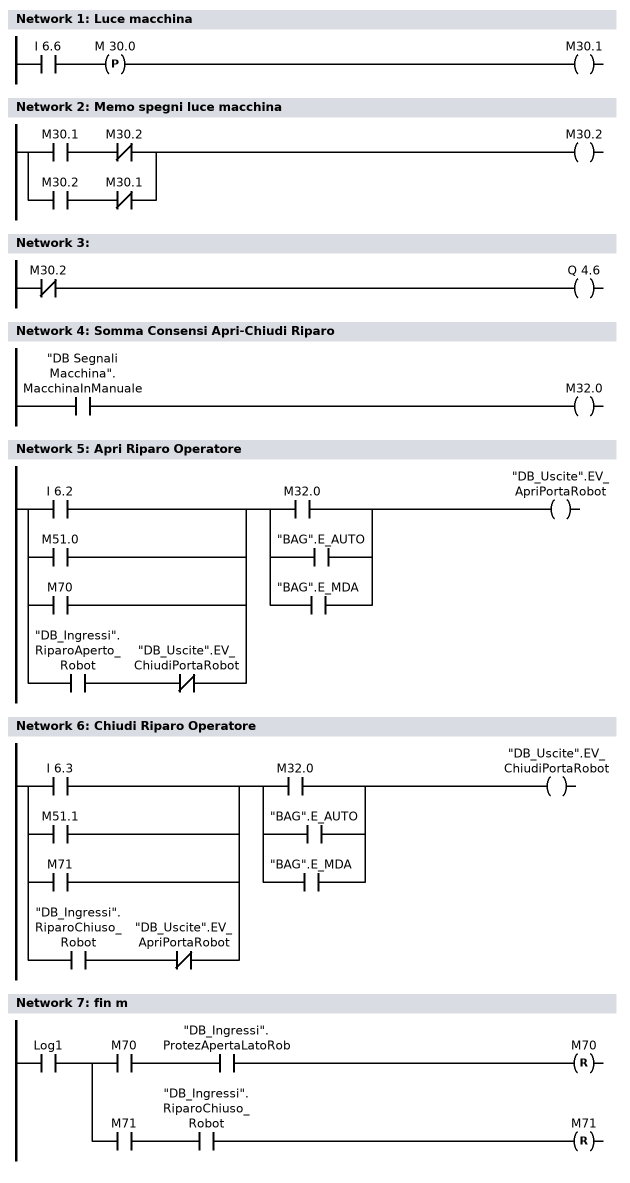
NETWORK
TITLE = Luce macchina
      A     I 6.6;
      FP    M 30.0;
      =     "M30.1";
NETWORK
TITLE = Memo spegni luce macchina
      A     "M30.1";
      AN    "M30.2";
      O;
      A     "M30.2";
      AN    "M30.1";
      =     "M30.2";
NETWORK
TITLE =
      AN    "M30.2";
      =     Q 4.6;
NETWORK
TITLE = Somma Consensi Apri-Chiudi Riparo
      A     "DB Segnali Macchina".MacchinaInManuale;
      =     "M32.0";
NETWORK
TITLE = Apri Riparo Operatore
      A(;
      O     I 6.2;
      O     "M51.0";
      O     "M70";
      O;
      A     "DB_Ingressi".RiparoAperto_Robot;
      AN    "DB_Uscite".EV_ChiudiPortaRobot;
      );
      A(;
      O     "M32.0";
      O     "BAG".E_AUTO;
      O     "BAG".E_MDA;
      );
      =     "DB_Uscite".EV_ApriPortaRobot;
NETWORK
TITLE = Chiudi Riparo Operatore
      A(;
      O     I 6.3;
      O     "M51.1";
      O     "M71";
      O;
      A     "DB_Ingressi".RiparoChiuso_Robot;
      AN    "DB_Uscite".EV_ApriPortaRobot;
      );
      A(;
      O     "M32.0";
      O     "BAG".E_AUTO;
      O     "BAG".E_MDA;
      );
      =     "DB_Uscite".EV_ChiudiPortaRobot;
NETWORK
TITLE = fin m
      A     "Log1";
      =     L 0.0;
      A     L 0.0;
      A     "M70";
      A     "DB_Ingressi".ProtezApertaLatoRob;
      R     "M70";
      A     L 0.0;
      A     "M71";
      A     "DB_Ingressi".RiparoChiuso_Robot;
      R     "M71";
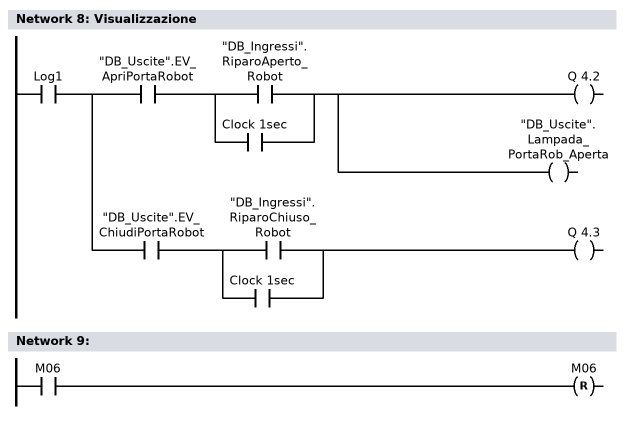
NETWORK
TITLE = Visualizzazione
      A     "Log1";
      =     L 0.0;
      A     L 0.0;
      A     "DB_Uscite".EV_ApriPortaRobot;
      A(;
      O     "DB_Ingressi".RiparoAperto_Robot;
      O     "Clock 1sec";
      );
      =     Q 4.2;
      =     "DB_Uscite".Lampada_PortaRob_Aperta;
      A     L 0.0;
      A     "DB_Uscite".EV_ChiudiPortaRobot;
      A(;
      O     "DB_Ingressi".RiparoChiuso_Robot;
      O     "Clock 1sec";
      );
      =     Q 4.3;
NETWORK
TITLE =
      A     "M06";
      R     "M06";
END_FUNCTION

FUNCTION "FC Modi Operativi" : VOID	// FC 112
TITLE = Seleziona modo da selettore
VERSION : 0.1
BEGIN
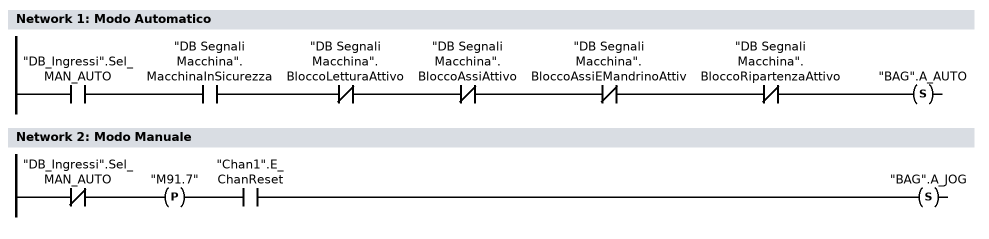
NETWORK
TITLE = Modo Automatico
      A     "DB_Ingressi".Sel_MAN_AUTO;
      A     "DB Segnali Macchina".MacchinaInSicurezza;
      AN    "DB Segnali Macchina".BloccoLetturaAttivo;
      AN    "DB Segnali Macchina".BloccoAssiAttivo;
      AN    "DB Segnali Macchina".BloccoAssiEMandrinoAttiv;
      AN    "DB Segnali Macchina".BloccoRipartenzaAttivo;
      S     "BAG".A_AUTO;
NETWORK
TITLE = Modo Manuale
      AN    "DB_Ingressi".Sel_MAN_AUTO;
      FP    "M91.7";
      A     "Chan1".E_ChanReset;
      S     "BAG".A_JOG;
END_FUNCTION

FUNCTION "FC Tastatura" : VOID	// FC 113
TITLE = Gestione Tastatura
VERSION : 0.1
BEGIN
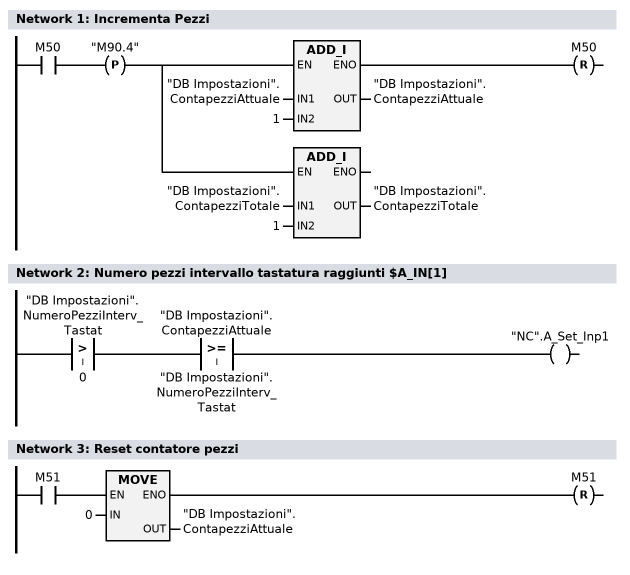
NETWORK
TITLE = Incrementa Pezzi
      A     "M50";
      FP    "M90.4";
      =     L 0.0;
      A     L 0.0;
      JNB   _001;
      L     "DB Impostazioni".ContapezziAttuale;
      L     1;
      +I;
      T     "DB Impostazioni".ContapezziAttuale;
      AN    OV;
      SAVE;
      CLR;
_001: A     BR;
      R     "M50";
      A     L 0.0;
      JNB   _002;
      L     "DB Impostazioni".ContapezziTotale;
      L     1;
      +I;
      T     "DB Impostazioni".ContapezziTotale;
_002: NOP   0;
NETWORK
TITLE = Numero pezzi intervallo tastatura raggiunti $A_IN[1]
      A(;
      L     "DB Impostazioni".NumeroPezziInterv_Tastat;
      L     0;
      >I;
      );
      A(;
      L     "DB Impostazioni".ContapezziAttuale;
      L     "DB Impostazioni".NumeroPezziInterv_Tastat;
      >=I;
      );
      =     "NC".A_Set_Inp1;
NETWORK
TITLE = Reset contatore pezzi
      A     "M51";
      JNB   _003;
      L     0;
      T     "DB Impostazioni".ContapezziAttuale;
      SET;
      SAVE;
      CLR;
_003: A     BR;
      R     "M51";
END_FUNCTION

FUNCTION "FC ComPCPlc" : VOID	// FC 114
VERSION : 0.1
VAR_TEMP
  Error : BOOL ;
  ErrCod : INT ;
END_VAR
BEGIN
NETWORK
TITLE = scambio dati robot
      CALL  "TIME_TCK" (
           RET_VAL                  := "PC<>PLC".ALIVE);
      A     "PC<>PLC".Pc_to_Plc.VivoPLC;
      =     "PC<>PLC".PLC_to_PC.PLC_Attivo;
NETWORK
TITLE = Scambio numero programma richiesto
      CALL  "Transfer" (
           $1                       := "PC<>PLC".Pc_to_Plc.ConsensoLetturaNrProg,
           $2                       := B#16#4,
           $3                       := "PC<>PLC".Pc_to_Plc.RichiestaTipo,
           $4                       := 0,
           $5                       := -1,
           $6                       := #Error,
           $7                       := #ErrCod);
      A     #Error;
      S     "DB Allarmi".Canale1.Feed_And_Read_Disable.A510125;
NETWORK
TITLE = info a robot
//-- macchina disponibile
      A     "DB_Ingressi".Sel_MAN_AUTO;
      A     "Chan1".E_ChanReset;
      AN    "Chan1".E_ProgRunn;
      A     "DB Segnali Macchina".MacchinaInSicurezza;
      =     "PC<>PLC".PLC_to_PC.ProntoPerComandi;
      A     "PC<>PLC".Pc_to_Plc.ConsensoLetturaNrProg;
      AN    #Error;
      =     "PC<>PLC".PLC_to_PC.NrProgrammaAcquisito;
      JCN   M999;
// echo nr programma
      L     "PC<>PLC".Pc_to_Plc.RichiestaTipo;
      T     "PC<>PLC".PLC_to_PC.DAto_01;
M999: NOP   0;
//-- riparo aperto
      A     "DB_Ingressi".RiparoAperto_Robot;
      =     "PC<>PLC".PLC_to_PC.RiparoAperto;
//-- riparo chiuso
      A     "DB_Ingressi".RiparoChiuso_Robot;
      =     "PC<>PLC".PLC_to_PC.RiparoChiuso;
//-- morsetta aperta
      A     "DB_Uscite".EV_ApriMorse;
      AN    "DB_Ingressi".PressPinzaMorsa;
      =     "PC<>PLC".PLC_to_PC.MorsaAperta;
//-- morsetta chiusa
      A     "DB_Uscite".EV_ChiudiMorse;
      A     "DB_Ingressi".PressPinzaMorsa;
      =     "PC<>PLC".PLC_to_PC.MorsaChiusa;
NETWORK
TITLE = // stati macchina
      A     "Chan1".E_ProgRunn;
      JC    M001;
      A     "Chan1".A_NCStartDisabl;
      JC    M002;
      A     "NC".A_EMERGENCY;
      JC    M003;
      A     "Chan1".E_ChanInterrupt;
      JC    M004;
      L     0;
      JU    END;
M001: NOP   0;	//programma in corso
      L     1;
      JU    END;
M002: NOP   0;	//start disabilitato
      L     2;
      JU    END;
M003: NOP   0;	//emergenza
      L     3;
      JU    END;
M004: NOP   0;
      L     4;
      JU    END;
      NOP   0;
      L     5;
      JU    END;
      NOP   0;
      L     6;
      JU    END;
      NOP   0;
      L     7;
      JU    END;
      NOP   0;
      L     8;
      JU    END;
      NOP   0;
      L     9;
      JU    END;
      NOP   0;
      L     10;
      JU    END;
END:  NOP   0;
      T     "PC<>PLC".PLC_to_PC.StatiMacchina;
NETWORK
TITLE = comandi da robot
//-- apertura riparo
      A     "PC<>PLC".Pc_to_Plc.ApriRiparo;
      FP    M 50.0;
      A     "PC<>PLC".PLC_to_PC.ProntoPerComandi;
      S     "M51.0";
      A     "PC<>PLC".PLC_to_PC.RiparoAperto;
      ON    "PC<>PLC".PLC_to_PC.ProntoPerComandi;
      R     "M51.0";
//-- chiusura riparo
      A     "PC<>PLC".Pc_to_Plc.ChiudiRiparo;
      FP    M 50.1;
      A     "PC<>PLC".PLC_to_PC.ProntoPerComandi;
      S     "M51.1";
      A     "PC<>PLC".PLC_to_PC.RiparoChiuso;
      ON    "PC<>PLC".PLC_to_PC.ProntoPerComandi;
      R     "M51.1";
//-- apertura morse
      A     "PC<>PLC".Pc_to_Plc.ApriMorsetta;
      FP    M 50.2;
      A     "PC<>PLC".PLC_to_PC.ProntoPerComandi;
      S     "M51.2";
      A     "PC<>PLC".PLC_to_PC.MorsaAperta;
      ON    "PC<>PLC".PLC_to_PC.ProntoPerComandi;
      R     "M51.2";
//-- chiusura morse
      A     "PC<>PLC".Pc_to_Plc.ChiudiMorsetta;
      FP    M 50.3;
      A     "PC<>PLC".PLC_to_PC.ProntoPerComandi;
      S     "M51.3";
      A     "PC<>PLC".PLC_to_PC.MorsaChiusa;
      ON    "PC<>PLC".PLC_to_PC.ProntoPerComandi;
      R     "M51.3";
//-- start ciclo
      A     "PC<>PLC".Pc_to_Plc.DatoBool_025;
      FP    M 50.4;
      S     "M51.4";
      A     "Chan1".E_ProgRunn;
      ON    "PC<>PLC".PLC_to_PC.ProntoPerComandi;
      R     "M51.4";
END_FUNCTION

FUNCTION "FC Intrefaccia Assi" : VOID	// FC 190
TITLE = TRASMISSIONE SEGNALI DI INTERFACCIA ASSE
AUTHOR : Asamec
NAME : itrf_ax
VERSION : 1.0
VAR_INPUT
  OVERR_ACT : BOOL ;	//OVERRIDE ATTIVO
  FUNZ_PUNT : BOOL ;	//SENSORE FUNZIONAMENTO A PUNTALINO
  RIC_FUNZ_PUNT : BOOL ;	//RICONOSC.FUNZIONAM. A PUNTALINO
  CONS_REGOL : BOOL ;	//CONSENSO REGOLATORE
  ABIL_IMP : BOOL ;	//ABILITAZIONE IMPULSI
  ATT_CAM_SW : BOOL ;	//ATTIVAZIONE CAMME SOFTWARE
  FC_SOFTWARE2_PIU : BOOL ;	//ATTIVAZIONE 2^ FC SOFTWARE PIU
  FC_SOFTWARE2_MENO : BOOL ;	//ATTIVAZIONE 2^ FC SOFTWARE MENO
  CONS_AVANZ : BOOL ;	//CONSENSO AVANZAMENTO ASSE
  OLTREC_PIU : BOOL ;	//OLTRECORSA HARDWARE POSITIVO
  CANC_PERC_RES : BOOL ;	//CANCELLAZIONE PERCORSO RESIDUO
  BLOC_AX : BOOL ;	//BLOCCAGGIO ASSE
  LIMIT_VEL : BOOL ;	//LIMITAZIONE VELOCITA'
  OVERR_RAP_ACT : BOOL ;	//OVERRIDE RAPIDO IN JOG ATTIVO
  JOG_STANDARD : BOOL ;
  JOG_MENO : BOOL ;	//MOVIMENTAZIONE IN JOG [-]
  JOG_PIU : BOOL ;	//MOVIMENTAZIONE IN JOG [+]
  VAL_INCR : BYTE ;	//VALORE IN INCREMENTALE
  OLTREC_MENO : BOOL ;	//OLTRECORSA HARDWARE NEGATIVO
  VAL_OVERR : BYTE ;	//VALORE OVERRIDE
  DB_INT_AX : INT ;	//DB DI INTERFACCIA PLC >> NCK
  SIST_MIS_1 : BOOL ;	//SISTEMA DI MISURAZIONE 1
  SIST_MIS_2 : BOOL ;	//SISTEMA DI MISURAZIONE 2
  AX_CAMME_REF : BOOL ;	//ASSE SU CAMME DI AZZERAMENTO
  PUNTO_REF_1 : BOOL ;	//1^ PUNTO DI RIFERIMENTO
END_VAR
VAR_OUTPUT
  MOV_AX : BOOL ;	//MOVIMENTAZIONE ASSE
  MOV_AX_MENO : BOOL ;	//MOVIMENTAZIONE ASSE IN DIREZIONE (-)
  MOV_AX_PIU : BOOL ;	//MOVIMENTAZIONE ASSE IN DIREZIONE (+)
  ASSE_FERMO : BOOL ;	//ASSE FERMO
  ASSE_AZZER : BOOL ;	//ASSE AZZERATO
END_VAR
VAR_TEMP
  DB_AX : INT ;	//DB DI INTERFACCIA ASSE
END_VAR
BEGIN
NETWORK
TITLE = APERTURA DB DI INTERFACCIA PLC >> NCK
      L     #DB_INT_AX;
      T     #DB_AX;
      OPN   DB [#DB_AX];
NETWORK
TITLE = SEGNALI VERSO NCK
      A     #OVERR_ACT;
      =     DBX 1.7;
      A     #FUNZ_PUNT;
      =     DBX 1.2;
      A     #RIC_FUNZ_PUNT;
      =     DBX 1.1;
      A     #ABIL_IMP;
      =     DBX 21.7;
      A     #ATT_CAM_SW;
      =     DBX 2.0;
      A     #FC_SOFTWARE2_PIU;
      =     DBX 12.3;
      A     #FC_SOFTWARE2_MENO;
      =     DBX 12.2;
      A     #CONS_AVANZ;
      =     DBX 4.3;
      A     #CANC_PERC_RES;
      =     DBX 2.2;
      A     #BLOC_AX;
      =     DBX 2.3;
      A     #LIMIT_VEL;
      =     DBX 3.6;
      A     #OVERR_RAP_ACT;
      =     DBX 4.5;
      AN    #JOG_STANDARD;
      JCN   NGS;
      A     #JOG_MENO;
      AN    #JOG_PIU;
      =     DBX 4.6;
      A     #JOG_PIU;
      AN    #JOG_MENO;
      =     DBX 4.7;
NGS:  NOP   0;
      A     #OLTREC_MENO;
      =     DBX 12.0;
      A     #OLTREC_PIU;
      =     DBX 12.1;
      A     #CONS_REGOL;
      =     DBX 2.1;
      A     #SIST_MIS_1;
      AN    #SIST_MIS_2;
      =     DBX 1.5;
      A     #SIST_MIS_2;
      AN    #SIST_MIS_1;
      =     DBX 1.6;
      A     #AX_CAMME_REF;
      =     DBX 12.7;
      A     #PUNTO_REF_1;
      =     DBX 2.4;
      L     #VAL_OVERR;
      OPN   DB [#DB_AX];
      T     DBB 0;
      L     #VAL_INCR;
      OPN   DB [#DB_AX];
      T     DBB 5;
NETWORK
TITLE = SEGNALI DA NCK
      A     DBX 64.6;
      O     DBX 64.7;
      =     #MOV_AX;
      A     DBX 64.6;
      =     #MOV_AX_MENO;
      A     DBX 64.7;
      =     #MOV_AX_PIU;
      A     DBX 61.4;
      =     #ASSE_FERMO;
      A     DBX 1.5;
      A     DBX 60.4;
      O;
      A     DBX 1.6;
      A     DBX 60.5;
      =     #ASSE_AZZER;
END_FUNCTION

FUNCTION "FC_Profibus_MM4" : VOID	// FC 191
AUTHOR : PROTEKNO
NAME : MM4
VERSION : 0.1
VAR_INPUT
  Periferic_Address : INT ;
  Drive_On_Off : BOOL ;
  Drive_Reversing : BOOL ;
  Drive_Fault_ACKN : BOOL ;
  Drive_F_Setpoint : REAL ;
END_VAR
VAR_OUTPUT
  Drive_in_operation : BOOL ;
  Drive_Fault_Active : BOOL ;
  Drive_Alarm_Active : BOOL ;
  Freno : BOOL ;
  Drive_F_Act : REAL ;
END_VAR
VAR_TEMP
  Address_E_A : DWORD ;
  SEND : STRUCT
   CW1 : UDT 91;
   f_setpoint : WORD ;
  END_STRUCT ;
  REC : STRUCT
   SW1 : UDT 92;
   f_act : WORD ;
  END_STRUCT ;
END_VAR
BEGIN
NETWORK
TITLE = Trasferimento indirizzo blocco;
      L     #Periferic_Address;
      SLD   3;
      T     #Address_E_A;
NETWORK
TITLE = Status word PZD MM4;
      L     PID [#Address_E_A];
      T     #REC;	//Status word MM4;
NETWORK
TITLE = control bit`s + setpoint
// ---------------------------------------
// IN-Variablen FC
// --------------------------------------
// PZD1 - Steuerwort 1                  // set single bit in the control word 1
      SET;	// set VKE=1
      =     #SEND.CW1.Bit_1;
      =     #SEND.CW1.Bit_2;
      =     #SEND.CW1.Bit_3;
      =     #SEND.CW1.Bit_4;
      =     #SEND.CW1.Bit_5;
      =     #SEND.CW1.Bit_6;
      =     #SEND.CW1.Bit_10;	// setpoint valid
      CLR;	// set VKE=0
      =     #SEND.CW1.Bit_8;
      =     #SEND.CW1.Bit_9;
      =     #SEND.CW1.Bit_12;
      =     #SEND.CW1.Bit_13;
      =     #SEND.CW1.Bit_14;
      =     #SEND.CW1.Bit_15;
      A     #Drive_On_Off;	// on / off ?
      =     #SEND.CW1.Bit_0;
      A     #Drive_Reversing;	// cw / cww ?
      =     #SEND.CW1.Bit_11;
      A     #Drive_Fault_ACKN;	// fault ackn.?
      =     #SEND.CW1.Bit_7;
//  
// PZD2 - Drehzahlsollwert
// gültiger Drehzahlsollwert zwischen 0.00-50 Hz
      L     #Drive_F_Setpoint;	// setpoint [Hz]
      L     0.000000e+00;
      <R;	// setpoinz >0Hz
      JC    N004;
      L     #Drive_F_Setpoint;
      L     7.500000e+01;
      >R;	// setpoint < 75Hz ?
      JC    N004;
      L     #Drive_F_Setpoint;
      L     1.000000e+02;	// 2-Nachkommastellen retten
      *R;
      RND;	//conversion of a 32-bit IEEE floating-point number to 32-bit integer
      L     24576;	// 16384 = 4000HEX = 50Hz
      *D;
      L     7500;
      /D;
      T     #SEND.f_setpoint;
N004: NOP   0;
NETWORK
TITLE = stateword + actual frequency 
// -------------------------------------
// OUT-Variablen FC                     
// -------------------------------------
// PZD 1 - Zustandswort
      A     #REC.SW1.Bit_2;
      =     #Drive_in_operation;
      A     #REC.SW1.Bit_3;
      =     #Drive_Fault_Active;
      A     #REC.SW1.Bit_7;
      =     #Drive_Alarm_Active;
      A     #REC.SW1.Bit_12;
      =     #Freno;
// PZD 2 - Drehzahlistwert
      L     #REC.f_act;
      ITD;
      DTR;
      L     5.000000e+01;	//16383= 4000HEX = 50Hz
      *R;
      L     1.638400e+04;
      /R;
      L     1.000000e+02;
      *R;
      TRUNC;
      ITD;
      DTR;
      L     1.000000e+02;
      /R;
      T     #Drive_F_Act;
NETWORK
TITLE = Control word PZD MM4;
      L     #SEND;	//Control word MM4;
      T     PQD [#Address_E_A];
      BE;
END_FUNCTION

// FC 200: know-how protected block, not included

// FC 1005: know-how protected block, not included

// FC 1006: know-how protected block, not included

// FC 1007: know-how protected block, not included

// FC 1008: know-how protected block, not included

// FC 1010: know-how protected block, not included

DATA_BLOCK "DB Allarmi"	// DB 2
AUTHOR : Asamec
VERSION : 0.0
  STRUCT
   Canale1 : STRUCT
    Feed_Disable : STRUCT
     A510000 : BOOL ;	//Attenzione Manca Aria
     A510001 : BOOL ;	//Fungo Consolle Premuto
     A510002 : BOOL ;	//Fungo CN Premuto
     A510003 : BOOL ;	//Fungo Robot Premuto
     A510004 : BOOL ;	//Anomalia Circuito recupero olio refrigerante
     A510005 : BOOL ;
     A510006 : BOOL ;
     A510007 : BOOL ;
     A510008 : BOOL ;	//rotazione mandrino con pinza aperta
     A510009 : BOOL ;
     A510010 : BOOL ;
     A510011 : BOOL ;
     A510012 : BOOL ;
     A510013 : BOOL ;
     A510014 : BOOL ;
     A510015 : BOOL ;
    END_STRUCT ;
    Feed_And_Read_Disable : STRUCT
     A510100 : BOOL ;	//Errore Tastatore Renishaw
     A510101 : BOOL ;	//Time-Out Funzione M
     A510102 : BOOL ;	//Time-Out Chiudi pinza Mandrino
     A510103 : BOOL ;	//Time-Out Apri pinza Mandrino
     A510104 : BOOL ;	//Termico Lubrificazione
     A510105 : BOOL ;	//Termico Centralina Idraulica
     A510106 : BOOL ;	//Termico Raffreddamento Centralina Idraulica
     A510107 : BOOL ;	//Termico Filtro Drives
     A510108 : BOOL ;	//Anomalia sensore Blocco-Sblocco Utensile
     A510109 : BOOL ;	//Anomalia Freno Asse A
     A510110 : BOOL ;	//Anomalia Freno Asse B
     A510111 : BOOL ;	//Pressione mandrino insufficiente
     A510112 : BOOL ;	//Pressione portamola insufficiente
     A510113 : BOOL ;	//Pressione portapezzo insufficiente
     A510114 : BOOL ;	//Termico Intervenuto Pompa Travaso
     A510115 : BOOL ;	//Anomalia Pompa Travaso (tempo massimo superato)
     A510116 : BOOL ;	//Anomalia Livello minimo vasca refrigerante
     A510117 : BOOL ;	//Anomalia Livello presenza olio vasca refrigerante
     A510118 : BOOL ;	//Probabile guasto livello massimo vasca refrigerante
     A510119 : BOOL ;	//Livello Massimo Refrigerante Vasca Interna
     A510120 : BOOL ;	//3 Tentativi ripristino refrigerante falliti
     A510121 : BOOL ;	//Anomalia Valvola refrigerante 1
     A510122 : BOOL ;	//Anomalia Valvola refrigerante 2
     A510123 : BOOL ;	//Termico Intervento Pompa Refrigerante
     A510124 : BOOL ;	//Richiesta di Start con ripari aperti
     A510125 : BOOL ;	//Attenzione si è verificato un errore di comunicazione tra PLC e NC
     A510126 : BOOL ;
     A510127 : BOOL ;
     A510128 : BOOL ;
     A510129 : BOOL ;
     A510130 : BOOL ;
     A510131 : BOOL ;
    END_STRUCT ;
    Read_Disable : STRUCT
     A510200 : BOOL ;
     A510201 : BOOL ;	//Anomalia Flussostato X
     A510202 : BOOL ;	//Anomalia Flussostato Y
     A510203 : BOOL ;	//Anomalia Flussostato Z
     A510204 : BOOL ;	//Anomalia Flussostato A
     A510205 : BOOL ;	//Anomalia Flussostato B
     A510206 : BOOL ;	//Anomalia Flussostato Elettromandrino
     A510207 : BOOL ;	//Anomalia Flussostato Rettifica Mole
     A510208 : BOOL ;	//Anomalia Flussostato 8
     A510209 : BOOL ;	//Allarme Termico motore raffreddamento
     A510210 : BOOL ;	//Anomalia Inverter Mandrino Diamantatura
     A510211 : BOOL ;	//Fault rilevato su mandrino diamantatura
     A510212 : BOOL ;
     A510213 : BOOL ;
     A510214 : BOOL ;
     A510215 : BOOL ;
     A510216 : BOOL ;	//Funzione M Attiva
     A510217 : BOOL ;
     A510218 : BOOL ;
     A510219 : BOOL ;
     A510220 : BOOL ;
     A510221 : BOOL ;
     A510222 : BOOL ;
     A510223 : BOOL ;
     A510224 : BOOL ;
     A510225 : BOOL ;
     A510226 : BOOL ;
     A510227 : BOOL ;
     A510228 : BOOL ;
     A510229 : BOOL ;
     A510230 : BOOL ;
     A510231 : BOOL ;
    END_STRUCT ;
    Start_Disable : STRUCT
     A510300 : BOOL ;	//Anomalia Lubrificazione Guide assi Lineari
     A510301 : BOOL ;
     A510302 : BOOL ;
     A510303 : BOOL ;
     A510304 : BOOL ;
     A510305 : BOOL ;
     A510306 : BOOL ;
     A510307 : BOOL ;
     A510308 : BOOL ;
     A510309 : BOOL ;
     A510310 : BOOL ;
     A510311 : BOOL ;
     A510312 : BOOL ;
     A510313 : BOOL ;
     A510314 : BOOL ;
     A510315 : BOOL ;
    END_STRUCT ;
    Feed_Stop_Asse_GEO1 : STRUCT
     A511100 : BOOL ;
     A511101 : BOOL ;
     A511102 : BOOL ;
     A511103 : BOOL ;
     A511104 : BOOL ;
     A511105 : BOOL ;
     A511106 : BOOL ;
     A511107 : BOOL ;
     A511108 : BOOL ;
     A511109 : BOOL ;
     A511110 : BOOL ;
     A511111 : BOOL ;
     A511112 : BOOL ;
     A511113 : BOOL ;
     A511114 : BOOL ;
     A511115 : BOOL ;
    END_STRUCT ;
    Feed_Stop_Asse_GEO2 : STRUCT
     A511200 : BOOL ;
     A511201 : BOOL ;
     A511202 : BOOL ;
     A511203 : BOOL ;
     A511204 : BOOL ;
     A511205 : BOOL ;
     A511206 : BOOL ;
     A511207 : BOOL ;
     A511208 : BOOL ;
     A511209 : BOOL ;
     A511210 : BOOL ;
     A511211 : BOOL ;
     A511212 : BOOL ;
     A511213 : BOOL ;
     A511214 : BOOL ;
     A511215 : BOOL ;
    END_STRUCT ;
    Feed_Stop_Asse_GEO3 : STRUCT
     A511300 : BOOL ;
     A511301 : BOOL ;
     A511302 : BOOL ;
     A511303 : BOOL ;
     A511304 : BOOL ;
     A511305 : BOOL ;
     A511306 : BOOL ;
     A511307 : BOOL ;
     A511308 : BOOL ;
     A511309 : BOOL ;
     A511310 : BOOL ;
     A511311 : BOOL ;
     A511312 : BOOL ;
     A511313 : BOOL ;
     A511314 : BOOL ;
     A511315 : BOOL ;
    END_STRUCT ;
   END_STRUCT ;
   Canale2 : STRUCT
    Feed_Disale : STRUCT
     A510000 : BOOL ;
     A510001 : BOOL ;
     A510002 : BOOL ;
     A510003 : BOOL ;
     A510004 : BOOL ;
     A510005 : BOOL ;
     A510006 : BOOL ;
     A510007 : BOOL ;
     A510008 : BOOL ;
     A510009 : BOOL ;
     A510010 : BOOL ;
     A510011 : BOOL ;
     A510012 : BOOL ;
     A510013 : BOOL ;
     A510014 : BOOL ;
     A510015 : BOOL ;
    END_STRUCT ;
    Feed_And_Read_Disable : STRUCT
     A510100 : BOOL ;
     A510101 : BOOL ;
     A510102 : BOOL ;
     A510103 : BOOL ;
     A510104 : BOOL ;
     A510105 : BOOL ;
     A510106 : BOOL ;
     A510107 : BOOL ;
     A510108 : BOOL ;
     A510109 : BOOL ;
     A510110 : BOOL ;
     A510111 : BOOL ;
     A510112 : BOOL ;
     A510113 : BOOL ;
     A510114 : BOOL ;
     A510115 : BOOL ;
     A510116 : BOOL ;
     A510117 : BOOL ;
     A510118 : BOOL ;
     A510119 : BOOL ;
     A510120 : BOOL ;
     A510121 : BOOL ;
     A510122 : BOOL ;
     A510123 : BOOL ;
     A510124 : BOOL ;
     A510125 : BOOL ;
     A510126 : BOOL ;
     A510127 : BOOL ;
     A510128 : BOOL ;
     A510129 : BOOL ;
     A510130 : BOOL ;
     A510131 : BOOL ;
    END_STRUCT ;
    Read_Disable : STRUCT
     A520000 : BOOL ;
     A520001 : BOOL ;
     A520002 : BOOL ;
     A520003 : BOOL ;
     A520004 : BOOL ;
     A520005 : BOOL ;
     A520006 : BOOL ;
     A520007 : BOOL ;
     A520008 : BOOL ;
     A520009 : BOOL ;
     A520010 : BOOL ;
     A520011 : BOOL ;
     A520012 : BOOL ;
     A520013 : BOOL ;
     A520014 : BOOL ;
     A520015 : BOOL ;
     A520016 : BOOL ;
     A520017 : BOOL ;
     A520018 : BOOL ;
     A520019 : BOOL ;
     A520020 : BOOL ;
     A520021 : BOOL ;
     A520022 : BOOL ;
     A520023 : BOOL ;
     A520024 : BOOL ;
     A520025 : BOOL ;
     A520026 : BOOL ;
     A520027 : BOOL ;
     A520028 : BOOL ;
     A520029 : BOOL ;
     A520030 : BOOL ;
     A520031 : BOOL ;
    END_STRUCT ;
    Start_Disable : STRUCT
     A530000 : BOOL ;
     A530001 : BOOL ;
     A530002 : BOOL ;
     A530003 : BOOL ;
     A530004 : BOOL ;
     A530005 : BOOL ;
     A530006 : BOOL ;
     A530007 : BOOL ;
     A530008 : BOOL ;
     A530009 : BOOL ;
     A530010 : BOOL ;
     A530011 : BOOL ;
     A530012 : BOOL ;
     A530013 : BOOL ;
     A530014 : BOOL ;
     A530015 : BOOL ;
    END_STRUCT ;
    Feed_Stop_Asse_GEO1 : STRUCT
     A511100 : BOOL ;
     A511101 : BOOL ;
     A511102 : BOOL ;
     A511103 : BOOL ;
     A511104 : BOOL ;
     A511105 : BOOL ;
     A511106 : BOOL ;
     A511107 : BOOL ;
     A511108 : BOOL ;
     A511109 : BOOL ;
     A511110 : BOOL ;
     A511111 : BOOL ;
     A511112 : BOOL ;
     A511113 : BOOL ;
     A511114 : BOOL ;
     A511115 : BOOL ;
    END_STRUCT ;
    Feed_Stop_Asse_GEO2 : STRUCT
     A511200 : BOOL ;
     A511201 : BOOL ;
     A511202 : BOOL ;
     A511203 : BOOL ;
     A511204 : BOOL ;
     A511205 : BOOL ;
     A511206 : BOOL ;
     A511207 : BOOL ;
     A511208 : BOOL ;
     A511209 : BOOL ;
     A511210 : BOOL ;
     A511211 : BOOL ;
     A511212 : BOOL ;
     A511213 : BOOL ;
     A511214 : BOOL ;
     A511215 : BOOL ;
    END_STRUCT ;
    Feed_Stop_Asse_GEO3 : STRUCT
     A511300 : BOOL ;
     A511301 : BOOL ;
     A511302 : BOOL ;
     A511303 : BOOL ;
     A511304 : BOOL ;
     A511305 : BOOL ;
     A511306 : BOOL ;
     A511307 : BOOL ;
     A511308 : BOOL ;
     A511309 : BOOL ;
     A511310 : BOOL ;
     A511311 : BOOL ;
     A511312 : BOOL ;
     A511313 : BOOL ;
     A511314 : BOOL ;
     A511315 : BOOL ;
    END_STRUCT ;
   END_STRUCT ;
   Canale3 : STRUCT
    Feed_Disale : STRUCT
     A510000 : BOOL ;
     A510001 : BOOL ;
     A510002 : BOOL ;
     A510003 : BOOL ;
     A510004 : BOOL ;
     A510005 : BOOL ;
     A510006 : BOOL ;
     A510007 : BOOL ;
     A510008 : BOOL ;
     A510009 : BOOL ;
     A510010 : BOOL ;
     A510011 : BOOL ;
     A510012 : BOOL ;
     A510013 : BOOL ;
     A510014 : BOOL ;
     A510015 : BOOL ;
    END_STRUCT ;
    Feed_And_Read_Disable : STRUCT
     A510100 : BOOL ;
     A510101 : BOOL ;
     A510102 : BOOL ;
     A510103 : BOOL ;
     A510104 : BOOL ;
     A510105 : BOOL ;
     A510106 : BOOL ;
     A510107 : BOOL ;
     A510108 : BOOL ;
     A510109 : BOOL ;
     A510110 : BOOL ;
     A510111 : BOOL ;
     A510112 : BOOL ;
     A510113 : BOOL ;
     A510114 : BOOL ;
     A510115 : BOOL ;
     A510116 : BOOL ;
     A510117 : BOOL ;
     A510118 : BOOL ;
     A510119 : BOOL ;
     A510120 : BOOL ;
     A510121 : BOOL ;
     A510122 : BOOL ;
     A510123 : BOOL ;
     A510124 : BOOL ;
     A510125 : BOOL ;
     A510126 : BOOL ;
     A510127 : BOOL ;
     A510128 : BOOL ;
     A510129 : BOOL ;
     A510130 : BOOL ;
     A510131 : BOOL ;
    END_STRUCT ;
    Read_Disable : STRUCT
     A520000 : BOOL ;
     A520001 : BOOL ;
     A520002 : BOOL ;
     A520003 : BOOL ;
     A520004 : BOOL ;
     A520005 : BOOL ;
     A520006 : BOOL ;
     A520007 : BOOL ;
     A520008 : BOOL ;
     A520009 : BOOL ;
     A520010 : BOOL ;
     A520011 : BOOL ;
     A520012 : BOOL ;
     A520013 : BOOL ;
     A520014 : BOOL ;
     A520015 : BOOL ;
     A520016 : BOOL ;
     A520017 : BOOL ;
     A520018 : BOOL ;
     A520019 : BOOL ;
     A520020 : BOOL ;
     A520021 : BOOL ;
     A520022 : BOOL ;
     A520023 : BOOL ;
     A520024 : BOOL ;
     A520025 : BOOL ;
     A520026 : BOOL ;
     A520027 : BOOL ;
     A520028 : BOOL ;
     A520029 : BOOL ;
     A520030 : BOOL ;
     A520031 : BOOL ;
    END_STRUCT ;
    Start_Disable : STRUCT
     A530000 : BOOL ;
     A530001 : BOOL ;
     A530002 : BOOL ;
     A530003 : BOOL ;
     A530004 : BOOL ;
     A530005 : BOOL ;
     A530006 : BOOL ;
     A530007 : BOOL ;
     A530008 : BOOL ;
     A530009 : BOOL ;
     A530010 : BOOL ;
     A530011 : BOOL ;
     A530012 : BOOL ;
     A530013 : BOOL ;
     A530014 : BOOL ;
     A530015 : BOOL ;
    END_STRUCT ;
    Feed_Stop_Asse_GEO1 : STRUCT
     A511100 : BOOL ;
     A511101 : BOOL ;
     A511102 : BOOL ;
     A511103 : BOOL ;
     A511104 : BOOL ;
     A511105 : BOOL ;
     A511106 : BOOL ;
     A511107 : BOOL ;
     A511108 : BOOL ;
     A511109 : BOOL ;
     A511110 : BOOL ;
     A511111 : BOOL ;
     A511112 : BOOL ;
     A511113 : BOOL ;
     A511114 : BOOL ;
     A511115 : BOOL ;
    END_STRUCT ;
    Feed_Stop_Asse_GEO2 : STRUCT
     A511200 : BOOL ;
     A511201 : BOOL ;
     A511202 : BOOL ;
     A511203 : BOOL ;
     A511204 : BOOL ;
     A511205 : BOOL ;
     A511206 : BOOL ;
     A511207 : BOOL ;
     A511208 : BOOL ;
     A511209 : BOOL ;
     A511210 : BOOL ;
     A511211 : BOOL ;
     A511212 : BOOL ;
     A511213 : BOOL ;
     A511214 : BOOL ;
     A511215 : BOOL ;
    END_STRUCT ;
    Feed_Stop_Asse_GEO3 : STRUCT
     A511300 : BOOL ;
     A511301 : BOOL ;
     A511302 : BOOL ;
     A511303 : BOOL ;
     A511304 : BOOL ;
     A511305 : BOOL ;
     A511306 : BOOL ;
     A511307 : BOOL ;
     A511308 : BOOL ;
     A511309 : BOOL ;
     A511310 : BOOL ;
     A511311 : BOOL ;
     A511312 : BOOL ;
     A511313 : BOOL ;
     A511314 : BOOL ;
     A511315 : BOOL ;
    END_STRUCT ;
   END_STRUCT ;
   Canale4 : STRUCT
    Feed_Disale : STRUCT
     A510000 : BOOL ;
     A510001 : BOOL ;
     A510002 : BOOL ;
     A510003 : BOOL ;
     A510004 : BOOL ;
     A510005 : BOOL ;
     A510006 : BOOL ;
     A510007 : BOOL ;
     A510008 : BOOL ;
     A510009 : BOOL ;
     A510010 : BOOL ;
     A510011 : BOOL ;
     A510012 : BOOL ;
     A510013 : BOOL ;
     A510014 : BOOL ;
     A510015 : BOOL ;
    END_STRUCT ;
    Feed_And_Read_Disable : STRUCT
     A510100 : BOOL ;
     A510101 : BOOL ;
     A510102 : BOOL ;
     A510103 : BOOL ;
     A510104 : BOOL ;
     A510105 : BOOL ;
     A510106 : BOOL ;
     A510107 : BOOL ;
     A510108 : BOOL ;
     A510109 : BOOL ;
     A510110 : BOOL ;
     A510111 : BOOL ;
     A510112 : BOOL ;
     A510113 : BOOL ;
     A510114 : BOOL ;
     A510115 : BOOL ;
     A510116 : BOOL ;
     A510117 : BOOL ;
     A510118 : BOOL ;
     A510119 : BOOL ;
     A510120 : BOOL ;
     A510121 : BOOL ;
     A510122 : BOOL ;
     A510123 : BOOL ;
     A510124 : BOOL ;
     A510125 : BOOL ;
     A510126 : BOOL ;
     A510127 : BOOL ;
     A510128 : BOOL ;
     A510129 : BOOL ;
     A510130 : BOOL ;
     A510131 : BOOL ;
    END_STRUCT ;
    Read_Disable : STRUCT
     A520000 : BOOL ;	//Funzione M in corso...
     A520001 : BOOL ;
     A520002 : BOOL ;
     A520003 : BOOL ;
     A520004 : BOOL ;
     A520005 : BOOL ;
     A520006 : BOOL ;
     A520007 : BOOL ;
     A520008 : BOOL ;
     A520009 : BOOL ;
     A520010 : BOOL ;
     A520011 : BOOL ;
     A520012 : BOOL ;
     A520013 : BOOL ;
     A520014 : BOOL ;
     A520015 : BOOL ;
     A520016 : BOOL ;
     A520017 : BOOL ;
     A520018 : BOOL ;
     A520019 : BOOL ;
     A520020 : BOOL ;
     A520021 : BOOL ;
     A520022 : BOOL ;
     A520023 : BOOL ;
     A520024 : BOOL ;
     A520025 : BOOL ;
     A520026 : BOOL ;
     A520027 : BOOL ;
     A520028 : BOOL ;
     A520029 : BOOL ;
     A520030 : BOOL ;
     A520031 : BOOL ;
    END_STRUCT ;
    Start_Disable : STRUCT
     A530000 : BOOL ;
     A530001 : BOOL ;
     A530002 : BOOL ;
     A530003 : BOOL ;
     A530004 : BOOL ;
     A530005 : BOOL ;
     A530006 : BOOL ;
     A530007 : BOOL ;
     A530008 : BOOL ;
     A530009 : BOOL ;
     A530010 : BOOL ;
     A530011 : BOOL ;
     A530012 : BOOL ;
     A530013 : BOOL ;
     A530014 : BOOL ;
     A530015 : BOOL ;
    END_STRUCT ;
    Feed_Stop_Asse_GEO1 : STRUCT
     A511100 : BOOL ;
     A511101 : BOOL ;
     A511102 : BOOL ;
     A511103 : BOOL ;
     A511104 : BOOL ;
     A511105 : BOOL ;
     A511106 : BOOL ;
     A511107 : BOOL ;
     A511108 : BOOL ;
     A511109 : BOOL ;
     A511110 : BOOL ;
     A511111 : BOOL ;
     A511112 : BOOL ;
     A511113 : BOOL ;
     A511114 : BOOL ;
     A511115 : BOOL ;
    END_STRUCT ;
    Feed_Stop_Asse_GEO2 : STRUCT
     A511200 : BOOL ;
     A511201 : BOOL ;
     A511202 : BOOL ;
     A511203 : BOOL ;
     A511204 : BOOL ;
     A511205 : BOOL ;
     A511206 : BOOL ;
     A511207 : BOOL ;
     A511208 : BOOL ;
     A511209 : BOOL ;
     A511210 : BOOL ;
     A511211 : BOOL ;
     A511212 : BOOL ;
     A511213 : BOOL ;
     A511214 : BOOL ;
     A511215 : BOOL ;
    END_STRUCT ;
    Feed_Stop_Asse_GEO3 : STRUCT
     A511300 : BOOL ;
     A511301 : BOOL ;
     A511302 : BOOL ;
     A511303 : BOOL ;
     A511304 : BOOL ;
     A511305 : BOOL ;
     A511306 : BOOL ;
     A511307 : BOOL ;
     A511308 : BOOL ;
     A511309 : BOOL ;
     A511310 : BOOL ;
     A511311 : BOOL ;
     A511312 : BOOL ;
     A511313 : BOOL ;
     A511314 : BOOL ;
     A511315 : BOOL ;
    END_STRUCT ;
   END_STRUCT ;
   Canale5 : STRUCT
    Feed_Disale : STRUCT
     A510000 : BOOL ;
     A510001 : BOOL ;
     A510002 : BOOL ;
     A510003 : BOOL ;
     A510004 : BOOL ;
     A510005 : BOOL ;
     A510006 : BOOL ;
     A510007 : BOOL ;
     A510008 : BOOL ;
     A510009 : BOOL ;
     A510010 : BOOL ;
     A510011 : BOOL ;
     A510012 : BOOL ;
     A510013 : BOOL ;
     A510014 : BOOL ;
     A510015 : BOOL ;
    END_STRUCT ;
    Feed_And_Read_Disable : STRUCT
     A510100 : BOOL ;
     A510101 : BOOL ;
     A510102 : BOOL ;
     A510103 : BOOL ;
     A510104 : BOOL ;
     A510105 : BOOL ;
     A510106 : BOOL ;
     A510107 : BOOL ;
     A510108 : BOOL ;
     A510109 : BOOL ;
     A510110 : BOOL ;
     A510111 : BOOL ;
     A510112 : BOOL ;
     A510113 : BOOL ;
     A510114 : BOOL ;
     A510115 : BOOL ;
     A510116 : BOOL ;
     A510117 : BOOL ;
     A510118 : BOOL ;
     A510119 : BOOL ;
     A510120 : BOOL ;
     A510121 : BOOL ;
     A510122 : BOOL ;
     A510123 : BOOL ;
     A510124 : BOOL ;
     A510125 : BOOL ;
     A510126 : BOOL ;
     A510127 : BOOL ;
     A510128 : BOOL ;
     A510129 : BOOL ;
     A510130 : BOOL ;
     A510131 : BOOL ;
    END_STRUCT ;
    Read_Disable : STRUCT
     A520000 : BOOL ;
     A520001 : BOOL ;
     A520002 : BOOL ;
     A520003 : BOOL ;
     A520004 : BOOL ;
     A520005 : BOOL ;
     A520006 : BOOL ;
     A520007 : BOOL ;
     A520008 : BOOL ;
     A520009 : BOOL ;
     A520010 : BOOL ;
     A520011 : BOOL ;
     A520012 : BOOL ;
     A520013 : BOOL ;
     A520014 : BOOL ;
     A520015 : BOOL ;
     A520016 : BOOL ;
     A520017 : BOOL ;
     A520018 : BOOL ;
     A520019 : BOOL ;
     A520020 : BOOL ;
     A520021 : BOOL ;
     A520022 : BOOL ;
     A520023 : BOOL ;
     A520024 : BOOL ;
     A520025 : BOOL ;
     A520026 : BOOL ;
     A520027 : BOOL ;
     A520028 : BOOL ;
     A520029 : BOOL ;
     A520030 : BOOL ;
     A520031 : BOOL ;
    END_STRUCT ;
    Start_Disable : STRUCT
     A530000 : BOOL ;
     A530001 : BOOL ;
     A530002 : BOOL ;
     A530003 : BOOL ;
     A530004 : BOOL ;
     A530005 : BOOL ;
     A530006 : BOOL ;
     A530007 : BOOL ;
     A530008 : BOOL ;
     A530009 : BOOL ;
     A530010 : BOOL ;
     A530011 : BOOL ;
     A530012 : BOOL ;
     A530013 : BOOL ;
     A530014 : BOOL ;
     A530015 : BOOL ;
    END_STRUCT ;
    Feed_Stop_Asse_GEO1 : STRUCT
     A511100 : BOOL ;
     A511101 : BOOL ;
     A511102 : BOOL ;
     A511103 : BOOL ;
     A511104 : BOOL ;
     A511105 : BOOL ;
     A511106 : BOOL ;
     A511107 : BOOL ;
     A511108 : BOOL ;
     A511109 : BOOL ;
     A511110 : BOOL ;
     A511111 : BOOL ;
     A511112 : BOOL ;
     A511113 : BOOL ;
     A511114 : BOOL ;
     A511115 : BOOL ;
    END_STRUCT ;
    Feed_Stop_Asse_GEO2 : STRUCT
     A511200 : BOOL ;
     A511201 : BOOL ;
     A511202 : BOOL ;
     A511203 : BOOL ;
     A511204 : BOOL ;
     A511205 : BOOL ;
     A511206 : BOOL ;
     A511207 : BOOL ;
     A511208 : BOOL ;
     A511209 : BOOL ;
     A511210 : BOOL ;
     A511211 : BOOL ;
     A511212 : BOOL ;
     A511213 : BOOL ;
     A511214 : BOOL ;
     A511215 : BOOL ;
    END_STRUCT ;
    Feed_Stop_Asse_GEO3 : STRUCT
     A511300 : BOOL ;
     A511301 : BOOL ;
     A511302 : BOOL ;
     A511303 : BOOL ;
     A511304 : BOOL ;
     A511305 : BOOL ;
     A511306 : BOOL ;
     A511307 : BOOL ;
     A511308 : BOOL ;
     A511309 : BOOL ;
     A511310 : BOOL ;
     A511311 : BOOL ;
     A511312 : BOOL ;
     A511313 : BOOL ;
     A511314 : BOOL ;
     A511315 : BOOL ;
    END_STRUCT ;
   END_STRUCT ;
   Canale6 : STRUCT
    Feed_Disale : STRUCT
     A510000 : BOOL ;
     A510001 : BOOL ;
     A510002 : BOOL ;
     A510003 : BOOL ;
     A510004 : BOOL ;
     A510005 : BOOL ;
     A510006 : BOOL ;
     A510007 : BOOL ;
     A510008 : BOOL ;
     A510009 : BOOL ;
     A510010 : BOOL ;
     A510011 : BOOL ;
     A510012 : BOOL ;
     A510013 : BOOL ;
     A510014 : BOOL ;
     A510015 : BOOL ;
    END_STRUCT ;
    Feed_And_Read_Disable : STRUCT
     A510100 : BOOL ;
     A510101 : BOOL ;
     A510102 : BOOL ;
     A510103 : BOOL ;
     A510104 : BOOL ;
     A510105 : BOOL ;
     A510106 : BOOL ;
     A510107 : BOOL ;
     A510108 : BOOL ;
     A510109 : BOOL ;
     A510110 : BOOL ;
     A510111 : BOOL ;
     A510112 : BOOL ;
     A510113 : BOOL ;
     A510114 : BOOL ;
     A510115 : BOOL ;
     A510116 : BOOL ;
     A510117 : BOOL ;
     A510118 : BOOL ;
     A510119 : BOOL ;
     A510120 : BOOL ;
     A510121 : BOOL ;
     A510122 : BOOL ;
     A510123 : BOOL ;
     A510124 : BOOL ;
     A510125 : BOOL ;
     A510126 : BOOL ;
     A510127 : BOOL ;
     A510128 : BOOL ;
     A510129 : BOOL ;
     A510130 : BOOL ;
     A510131 : BOOL ;
    END_STRUCT ;
    Read_Disable : STRUCT
     A520000 : BOOL ;
     A520001 : BOOL ;
     A520002 : BOOL ;
     A520003 : BOOL ;
     A520004 : BOOL ;
     A520005 : BOOL ;
     A520006 : BOOL ;
     A520007 : BOOL ;
     A520008 : BOOL ;
     A520009 : BOOL ;
     A520010 : BOOL ;
     A520011 : BOOL ;
     A520012 : BOOL ;
     A520013 : BOOL ;
     A520014 : BOOL ;
     A520015 : BOOL ;
     A520016 : BOOL ;
     A520017 : BOOL ;
     A520018 : BOOL ;
     A520019 : BOOL ;
     A520020 : BOOL ;
     A520021 : BOOL ;
     A520022 : BOOL ;
     A520023 : BOOL ;
     A520024 : BOOL ;
     A520025 : BOOL ;
     A520026 : BOOL ;
     A520027 : BOOL ;
     A520028 : BOOL ;
     A520029 : BOOL ;
     A520030 : BOOL ;
     A520031 : BOOL ;
    END_STRUCT ;
    Start_Disable : STRUCT
     A530000 : BOOL ;
     A530001 : BOOL ;
     A530002 : BOOL ;
     A530003 : BOOL ;
     A530004 : BOOL ;
     A530005 : BOOL ;
     A530006 : BOOL ;
     A530007 : BOOL ;
     A530008 : BOOL ;
     A530009 : BOOL ;
     A530010 : BOOL ;
     A530011 : BOOL ;
     A530012 : BOOL ;
     A530013 : BOOL ;
     A530014 : BOOL ;
     A530015 : BOOL ;
    END_STRUCT ;
    Feed_Stop_Asse_GEO1 : STRUCT
     A511100 : BOOL ;
     A511101 : BOOL ;
     A511102 : BOOL ;
     A511103 : BOOL ;
     A511104 : BOOL ;
     A511105 : BOOL ;
     A511106 : BOOL ;
     A511107 : BOOL ;
     A511108 : BOOL ;
     A511109 : BOOL ;
     A511110 : BOOL ;
     A511111 : BOOL ;
     A511112 : BOOL ;
     A511113 : BOOL ;
     A511114 : BOOL ;
     A511115 : BOOL ;
    END_STRUCT ;
    Feed_Stop_Asse_GEO2 : STRUCT
     A511200 : BOOL ;
     A511201 : BOOL ;
     A511202 : BOOL ;
     A511203 : BOOL ;
     A511204 : BOOL ;
     A511205 : BOOL ;
     A511206 : BOOL ;
     A511207 : BOOL ;
     A511208 : BOOL ;
     A511209 : BOOL ;
     A511210 : BOOL ;
     A511211 : BOOL ;
     A511212 : BOOL ;
     A511213 : BOOL ;
     A511214 : BOOL ;
     A511215 : BOOL ;
    END_STRUCT ;
    Feed_Stop_Asse_GEO3 : STRUCT
     A511300 : BOOL ;
     A511301 : BOOL ;
     A511302 : BOOL ;
     A511303 : BOOL ;
     A511304 : BOOL ;
     A511305 : BOOL ;
     A511306 : BOOL ;
     A511307 : BOOL ;
     A511308 : BOOL ;
     A511309 : BOOL ;
     A511310 : BOOL ;
     A511311 : BOOL ;
     A511312 : BOOL ;
     A511313 : BOOL ;
     A511314 : BOOL ;
     A511315 : BOOL ;
    END_STRUCT ;
   END_STRUCT ;
   Canale7 : STRUCT
    Feed_Disale : STRUCT
     A510000 : BOOL ;
     A510001 : BOOL ;
     A510002 : BOOL ;
     A510003 : BOOL ;
     A510004 : BOOL ;
     A510005 : BOOL ;
     A510006 : BOOL ;
     A510007 : BOOL ;
     A510008 : BOOL ;
     A510009 : BOOL ;
     A510010 : BOOL ;
     A510011 : BOOL ;
     A510012 : BOOL ;
     A510013 : BOOL ;
     A510014 : BOOL ;
     A510015 : BOOL ;
    END_STRUCT ;
    Feed_And_Read_Disable : STRUCT
     A510100 : BOOL ;
     A510101 : BOOL ;
     A510102 : BOOL ;
     A510103 : BOOL ;
     A510104 : BOOL ;
     A510105 : BOOL ;
     A510106 : BOOL ;
     A510107 : BOOL ;
     A510108 : BOOL ;
     A510109 : BOOL ;
     A510110 : BOOL ;
     A510111 : BOOL ;
     A510112 : BOOL ;
     A510113 : BOOL ;
     A510114 : BOOL ;
     A510115 : BOOL ;
     A510116 : BOOL ;
     A510117 : BOOL ;
     A510118 : BOOL ;
     A510119 : BOOL ;
     A510120 : BOOL ;
     A510121 : BOOL ;
     A510122 : BOOL ;
     A510123 : BOOL ;
     A510124 : BOOL ;
     A510125 : BOOL ;
     A510126 : BOOL ;
     A510127 : BOOL ;
     A510128 : BOOL ;
     A510129 : BOOL ;
     A510130 : BOOL ;
     A510131 : BOOL ;
    END_STRUCT ;
    Read_Disable : STRUCT
     A520000 : BOOL ;
     A520001 : BOOL ;
     A520002 : BOOL ;
     A520003 : BOOL ;
     A520004 : BOOL ;
     A520005 : BOOL ;
     A520006 : BOOL ;
     A520007 : BOOL ;
     A520008 : BOOL ;
     A520009 : BOOL ;
     A520010 : BOOL ;
     A520011 : BOOL ;
     A520012 : BOOL ;
     A520013 : BOOL ;
     A520014 : BOOL ;
     A520015 : BOOL ;
     A520016 : BOOL ;
     A520017 : BOOL ;
     A520018 : BOOL ;
     A520019 : BOOL ;
     A520020 : BOOL ;
     A520021 : BOOL ;
     A520022 : BOOL ;
     A520023 : BOOL ;
     A520024 : BOOL ;
     A520025 : BOOL ;
     A520026 : BOOL ;
     A520027 : BOOL ;
     A520028 : BOOL ;
     A520029 : BOOL ;
     A520030 : BOOL ;
     A520031 : BOOL ;
    END_STRUCT ;
    Start_Disable : STRUCT
     A530000 : BOOL ;
     A530001 : BOOL ;
     A530002 : BOOL ;
     A530003 : BOOL ;
     A530004 : BOOL ;
     A530005 : BOOL ;
     A530006 : BOOL ;
     A530007 : BOOL ;
     A530008 : BOOL ;
     A530009 : BOOL ;
     A530010 : BOOL ;
     A530011 : BOOL ;
     A530012 : BOOL ;
     A530013 : BOOL ;
     A530014 : BOOL ;
     A530015 : BOOL ;
    END_STRUCT ;
    Feed_Stop_Asse_GEO1 : STRUCT
     A511100 : BOOL ;
     A511101 : BOOL ;
     A511102 : BOOL ;
     A511103 : BOOL ;
     A511104 : BOOL ;
     A511105 : BOOL ;
     A511106 : BOOL ;
     A511107 : BOOL ;
     A511108 : BOOL ;
     A511109 : BOOL ;
     A511110 : BOOL ;
     A511111 : BOOL ;
     A511112 : BOOL ;
     A511113 : BOOL ;
     A511114 : BOOL ;
     A511115 : BOOL ;
    END_STRUCT ;
    Feed_Stop_Asse_GEO2 : STRUCT
     A511200 : BOOL ;
     A511201 : BOOL ;
     A511202 : BOOL ;
     A511203 : BOOL ;
     A511204 : BOOL ;
     A511205 : BOOL ;
     A511206 : BOOL ;
     A511207 : BOOL ;
     A511208 : BOOL ;
     A511209 : BOOL ;
     A511210 : BOOL ;
     A511211 : BOOL ;
     A511212 : BOOL ;
     A511213 : BOOL ;
     A511214 : BOOL ;
     A511215 : BOOL ;
    END_STRUCT ;
    Feed_Stop_Asse_GEO3 : STRUCT
     A511300 : BOOL ;
     A511301 : BOOL ;
     A511302 : BOOL ;
     A511303 : BOOL ;
     A511304 : BOOL ;
     A511305 : BOOL ;
     A511306 : BOOL ;
     A511307 : BOOL ;
     A511308 : BOOL ;
     A511309 : BOOL ;
     A511310 : BOOL ;
     A511311 : BOOL ;
     A511312 : BOOL ;
     A511313 : BOOL ;
     A511314 : BOOL ;
     A511315 : BOOL ;
    END_STRUCT ;
   END_STRUCT ;
   Canale8 : STRUCT
    Feed_Disale : STRUCT
     A510000 : BOOL ;
     A510001 : BOOL ;
     A510002 : BOOL ;
     A510003 : BOOL ;
     A510004 : BOOL ;
     A510005 : BOOL ;
     A510006 : BOOL ;
     A510007 : BOOL ;
     A510008 : BOOL ;
     A510009 : BOOL ;
     A510010 : BOOL ;
     A510011 : BOOL ;
     A510012 : BOOL ;
     A510013 : BOOL ;
     A510014 : BOOL ;
     A510015 : BOOL ;
    END_STRUCT ;
    Feed_And_Read_Disable : STRUCT
     A510100 : BOOL ;
     A510101 : BOOL ;
     A510102 : BOOL ;
     A510103 : BOOL ;
     A510104 : BOOL ;
     A510105 : BOOL ;
     A510106 : BOOL ;
     A510107 : BOOL ;
     A510108 : BOOL ;
     A510109 : BOOL ;
     A510110 : BOOL ;
     A510111 : BOOL ;
     A510112 : BOOL ;
     A510113 : BOOL ;
     A510114 : BOOL ;
     A510115 : BOOL ;
     A510116 : BOOL ;
     A510117 : BOOL ;
     A510118 : BOOL ;
     A510119 : BOOL ;
     A510120 : BOOL ;
     A510121 : BOOL ;
     A510122 : BOOL ;
     A510123 : BOOL ;
     A510124 : BOOL ;
     A510125 : BOOL ;
     A510126 : BOOL ;
     A510127 : BOOL ;
     A510128 : BOOL ;
     A510129 : BOOL ;
     A510130 : BOOL ;
     A510131 : BOOL ;
    END_STRUCT ;
    Read_Disable : STRUCT
     A520000 : BOOL ;
     A520001 : BOOL ;
     A520002 : BOOL ;
     A520003 : BOOL ;
     A520004 : BOOL ;
     A520005 : BOOL ;
     A520006 : BOOL ;
     A520007 : BOOL ;
     A520008 : BOOL ;
     A520009 : BOOL ;
     A520010 : BOOL ;
     A520011 : BOOL ;
     A520012 : BOOL ;
     A520013 : BOOL ;
     A520014 : BOOL ;
     A520015 : BOOL ;
     A520016 : BOOL ;
     A520017 : BOOL ;
     A520018 : BOOL ;
     A520019 : BOOL ;
     A520020 : BOOL ;
     A520021 : BOOL ;
     A520022 : BOOL ;
     A520023 : BOOL ;
     A520024 : BOOL ;
     A520025 : BOOL ;
     A520026 : BOOL ;
     A520027 : BOOL ;
     A520028 : BOOL ;
     A520029 : BOOL ;
     A520030 : BOOL ;
     A520031 : BOOL ;
    END_STRUCT ;
    Start_Disable : STRUCT
     A530000 : BOOL ;
     A530001 : BOOL ;
     A530002 : BOOL ;
     A530003 : BOOL ;
     A530004 : BOOL ;
     A530005 : BOOL ;
     A530006 : BOOL ;
     A530007 : BOOL ;
     A530008 : BOOL ;
     A530009 : BOOL ;
     A530010 : BOOL ;
     A530011 : BOOL ;
     A530012 : BOOL ;
     A530013 : BOOL ;
     A530014 : BOOL ;
     A530015 : BOOL ;
    END_STRUCT ;
    Feed_Stop_Asse_GEO1 : STRUCT
     A511100 : BOOL ;
     A511101 : BOOL ;
     A511102 : BOOL ;
     A511103 : BOOL ;
     A511104 : BOOL ;
     A511105 : BOOL ;
     A511106 : BOOL ;
     A511107 : BOOL ;
     A511108 : BOOL ;
     A511109 : BOOL ;
     A511110 : BOOL ;
     A511111 : BOOL ;
     A511112 : BOOL ;
     A511113 : BOOL ;
     A511114 : BOOL ;
     A511115 : BOOL ;
    END_STRUCT ;
    Feed_Stop_Asse_GEO2 : STRUCT
     A511200 : BOOL ;
     A511201 : BOOL ;
     A511202 : BOOL ;
     A511203 : BOOL ;
     A511204 : BOOL ;
     A511205 : BOOL ;
     A511206 : BOOL ;
     A511207 : BOOL ;
     A511208 : BOOL ;
     A511209 : BOOL ;
     A511210 : BOOL ;
     A511211 : BOOL ;
     A511212 : BOOL ;
     A511213 : BOOL ;
     A511214 : BOOL ;
     A511215 : BOOL ;
    END_STRUCT ;
    Feed_Stop_Asse_GEO3 : STRUCT
     A511300 : BOOL ;
     A511301 : BOOL ;
     A511302 : BOOL ;
     A511303 : BOOL ;
     A511304 : BOOL ;
     A511305 : BOOL ;
     A511306 : BOOL ;
     A511307 : BOOL ;
     A511308 : BOOL ;
     A511309 : BOOL ;
     A511310 : BOOL ;
     A511311 : BOOL ;
     A511312 : BOOL ;
     A511313 : BOOL ;
     A511314 : BOOL ;
     A511315 : BOOL ;
    END_STRUCT ;
   END_STRUCT ;
   Asse1_Feed_Stop : STRUCT
    A600100 : BOOL ;
    A600101 : BOOL ;
    A600102 : BOOL ;
    A600103 : BOOL ;
    A600104 : BOOL ;
    A600105 : BOOL ;
    A600106 : BOOL ;
    A600107 : BOOL ;
    A600108 : BOOL ;
    A600109 : BOOL ;
    A600110 : BOOL ;
    A600111 : BOOL ;
    A600112 : BOOL ;
    A600113 : BOOL ;
    A600114 : BOOL ;
    A600115 : BOOL ;
   END_STRUCT ;
   Asse2_Feed_Stop : STRUCT
    A600200 : BOOL ;
    A600201 : BOOL ;
    A600202 : BOOL ;
    A600203 : BOOL ;
    A600204 : BOOL ;
    A600205 : BOOL ;
    A600206 : BOOL ;
    A600207 : BOOL ;
    A600208 : BOOL ;
    A600209 : BOOL ;
    A600210 : BOOL ;
    A600211 : BOOL ;
    A600212 : BOOL ;
    A600213 : BOOL ;
    A600214 : BOOL ;
    A600215 : BOOL ;
   END_STRUCT ;
   Asse3_Feed_Stop : STRUCT
    A600300 : BOOL ;
    A600301 : BOOL ;
    A600302 : BOOL ;
    A600303 : BOOL ;
    A600304 : BOOL ;
    A600305 : BOOL ;
    A600306 : BOOL ;
    A600307 : BOOL ;
    A600308 : BOOL ;
    A600309 : BOOL ;
    A600310 : BOOL ;
    A600311 : BOOL ;
    A600312 : BOOL ;
    A600313 : BOOL ;
    A600314 : BOOL ;
    A600315 : BOOL ;
   END_STRUCT ;
   Asse4_Feed_Stop : STRUCT
    A600400 : BOOL ;
    A600401 : BOOL ;
    A600402 : BOOL ;
    A600403 : BOOL ;
    A600404 : BOOL ;
    A600405 : BOOL ;
    A600406 : BOOL ;
    A600407 : BOOL ;
    A600408 : BOOL ;
    A600409 : BOOL ;
    A600410 : BOOL ;
    A600411 : BOOL ;
    A600412 : BOOL ;
    A600413 : BOOL ;
    A600414 : BOOL ;
    A600415 : BOOL ;
   END_STRUCT ;
   Asse5_Feed_Stop : STRUCT
    A600500 : BOOL ;
    A600501 : BOOL ;
    A600502 : BOOL ;
    A600503 : BOOL ;
    A600504 : BOOL ;
    A600505 : BOOL ;
    A600506 : BOOL ;
    A600507 : BOOL ;
    A600508 : BOOL ;
    A600509 : BOOL ;
    A600510 : BOOL ;
    A600511 : BOOL ;
    A600512 : BOOL ;
    A600513 : BOOL ;
    A600514 : BOOL ;
    A600515 : BOOL ;
   END_STRUCT ;
   Asse6_Feed_Stop : STRUCT
    A600600 : BOOL ;
    A600601 : BOOL ;
    A600602 : BOOL ;
    A600603 : BOOL ;
    A600604 : BOOL ;
    A600605 : BOOL ;
    A600606 : BOOL ;
    A600607 : BOOL ;
    A600608 : BOOL ;
    A600609 : BOOL ;
    A600610 : BOOL ;
    A600611 : BOOL ;
    A600612 : BOOL ;
    A600613 : BOOL ;
    A600614 : BOOL ;
    A600615 : BOOL ;
   END_STRUCT ;
   Asse7_Feed_Stop : STRUCT
    A600700 : BOOL ;
    A600701 : BOOL ;
    A600702 : BOOL ;
    A600703 : BOOL ;
    A600704 : BOOL ;
    A600705 : BOOL ;
    A600706 : BOOL ;
    A600707 : BOOL ;
    A600708 : BOOL ;
    A600709 : BOOL ;
    A600710 : BOOL ;
    A600711 : BOOL ;
    A600712 : BOOL ;
    A600713 : BOOL ;
    A600714 : BOOL ;
    A600715 : BOOL ;
   END_STRUCT ;
   Asse8_Feed_Stop : STRUCT
    A600800 : BOOL ;
    A600801 : BOOL ;
    A600802 : BOOL ;
    A600803 : BOOL ;
    A600804 : BOOL ;
    A600805 : BOOL ;
    A600806 : BOOL ;
    A600807 : BOOL ;
    A600808 : BOOL ;
    A600809 : BOOL ;
    A600810 : BOOL ;
    A600811 : BOOL ;
    A600812 : BOOL ;
    A600813 : BOOL ;
    A600814 : BOOL ;
    A600815 : BOOL ;
   END_STRUCT ;
   Asse9_Feed_Stop : STRUCT
    A600900 : BOOL ;
    A600901 : BOOL ;
    A600902 : BOOL ;
    A600903 : BOOL ;
    A600904 : BOOL ;
    A600905 : BOOL ;
    A600906 : BOOL ;
    A600907 : BOOL ;
    A600908 : BOOL ;
    A600909 : BOOL ;
    A600910 : BOOL ;
    A600911 : BOOL ;
    A600912 : BOOL ;
    A600913 : BOOL ;
    A600914 : BOOL ;
    A600915 : BOOL ;
   END_STRUCT ;
   Asse10_Feed_Stop : STRUCT
    A601000 : BOOL ;
    A601001 : BOOL ;
    A601002 : BOOL ;
    A601003 : BOOL ;
    A601004 : BOOL ;
    A601005 : BOOL ;
    A601006 : BOOL ;
    A601007 : BOOL ;
    A601008 : BOOL ;
    A601009 : BOOL ;
    A601010 : BOOL ;
    A601011 : BOOL ;
    A601012 : BOOL ;
    A601013 : BOOL ;
    A601014 : BOOL ;
    A601015 : BOOL ;
   END_STRUCT ;
   Asse11_Feed_Stop : STRUCT
    A601100 : BOOL ;
    A601101 : BOOL ;
    A601102 : BOOL ;
    A601103 : BOOL ;
    A601104 : BOOL ;
    A601105 : BOOL ;
    A601106 : BOOL ;
    A601107 : BOOL ;
    A601108 : BOOL ;
    A601109 : BOOL ;
    A601110 : BOOL ;
    A601111 : BOOL ;
    A601112 : BOOL ;
    A601113 : BOOL ;
    A601114 : BOOL ;
    A601115 : BOOL ;
   END_STRUCT ;
   Asse12_Feed_Stop : STRUCT
    A601200 : BOOL ;
    A601201 : BOOL ;
    A601202 : BOOL ;
    A601203 : BOOL ;
    A601204 : BOOL ;
    A601205 : BOOL ;
    A601206 : BOOL ;
    A601207 : BOOL ;
    A601208 : BOOL ;
    A601209 : BOOL ;
    A601210 : BOOL ;
    A601211 : BOOL ;
    A601212 : BOOL ;
    A601213 : BOOL ;
    A601214 : BOOL ;
    A601215 : BOOL ;
   END_STRUCT ;
   Asse13_Feed_Stop : STRUCT
    A601300 : BOOL ;
    A601301 : BOOL ;
    A601302 : BOOL ;
    A601303 : BOOL ;
    A601304 : BOOL ;
    A601305 : BOOL ;
    A601306 : BOOL ;
    A601307 : BOOL ;
    A601308 : BOOL ;
    A601309 : BOOL ;
    A601310 : BOOL ;
    A601311 : BOOL ;
    A601312 : BOOL ;
    A601313 : BOOL ;
    A601314 : BOOL ;
    A601315 : BOOL ;
   END_STRUCT ;
   Asse14_Feed_Stop : STRUCT
    A601400 : BOOL ;
    A601401 : BOOL ;
    A601402 : BOOL ;
    A601403 : BOOL ;
    A601404 : BOOL ;
    A601405 : BOOL ;
    A601406 : BOOL ;
    A601407 : BOOL ;
    A601408 : BOOL ;
    A601409 : BOOL ;
    A601410 : BOOL ;
    A601411 : BOOL ;
    A601412 : BOOL ;
    A601413 : BOOL ;
    A601414 : BOOL ;
    A601415 : BOOL ;
   END_STRUCT ;
   Asse15_Feed_Stop : STRUCT
    A601500 : BOOL ;
    A601501 : BOOL ;
    A601502 : BOOL ;
    A601503 : BOOL ;
    A601504 : BOOL ;
    A601505 : BOOL ;
    A601506 : BOOL ;
    A601507 : BOOL ;
    A601508 : BOOL ;
    A601509 : BOOL ;
    A601510 : BOOL ;
    A601511 : BOOL ;
    A601512 : BOOL ;
    A601513 : BOOL ;
    A601514 : BOOL ;
    A601515 : BOOL ;
   END_STRUCT ;
   Asse16_Feed_Stop : STRUCT
    A601600 : BOOL ;
    A601601 : BOOL ;
    A601602 : BOOL ;
    A601603 : BOOL ;
    A601604 : BOOL ;
    A601605 : BOOL ;
    A601606 : BOOL ;
    A601607 : BOOL ;
    A601608 : BOOL ;
    A601609 : BOOL ;
    A601610 : BOOL ;
    A601611 : BOOL ;
    A601612 : BOOL ;
    A601613 : BOOL ;
    A601614 : BOOL ;
    A601615 : BOOL ;
   END_STRUCT ;
   Asse17_Feed_Stop : STRUCT
    A601700 : BOOL ;
    A601701 : BOOL ;
    A601702 : BOOL ;
    A601703 : BOOL ;
    A601704 : BOOL ;
    A601705 : BOOL ;
    A601706 : BOOL ;
    A601707 : BOOL ;
    A601708 : BOOL ;
    A601709 : BOOL ;
    A601710 : BOOL ;
    A601711 : BOOL ;
    A601712 : BOOL ;
    A601713 : BOOL ;
    A601714 : BOOL ;
    A601715 : BOOL ;
   END_STRUCT ;
   Asse18_Feed_Stop : STRUCT
    A601800 : BOOL ;
    A601801 : BOOL ;
    A601802 : BOOL ;
    A601803 : BOOL ;
    A601804 : BOOL ;
    A601805 : BOOL ;
    A601806 : BOOL ;
    A601807 : BOOL ;
    A601808 : BOOL ;
    A601809 : BOOL ;
    A601810 : BOOL ;
    A601811 : BOOL ;
    A601812 : BOOL ;
    A601813 : BOOL ;
    A601814 : BOOL ;
    A601815 : BOOL ;
   END_STRUCT ;
   Messaggi_User_Area0 : STRUCT
    A700000 : BOOL ;
    A700001 : BOOL ;	//Spindle Hold
    A700002 : BOOL ;	//Feed Hold
    A700003 : BOOL ;	//Riparo Aperto Operatore
    A700004 : BOOL ;	//Riparo Aperto Robot
    A700005 : BOOL ;	//Cancello Robot Aperto
    A700006 : BOOL ;	//Batteria scarica Renishaw
    A700007 : BOOL ;	//Attenzione livello massimo refrigerante
    A700008 : BOOL ;	//Attenzione Livello Massimo centralina idraulica
    A700009 : BOOL ;	//Attenzione Livello Basso Lubrificazione Guide assi Lineari
    A700010 : BOOL ;	//Attenzione rotazione mandrino non permessa con pinze aperte
    A700011 : BOOL ;
    A700012 : BOOL ;
    A700013 : BOOL ;
    A700014 : BOOL ;
    A700015 : BOOL ;
    A700016 : BOOL ;	//Extracorsa x+
    A700017 : BOOL ;	//Exrtacorsa x-
    A700018 : BOOL ;	//Extracorsa y +
    A700019 : BOOL ;	//Extracorsa y -
    A700020 : BOOL ;	//Extracorsa z +
    A700021 : BOOL ;	//Extracorsa z -
    A700022 : BOOL ;	//Erogazione Olio non possibile con porta aperta
    A700023 : BOOL ;
    A700024 : BOOL ;
    A700025 : BOOL ;
    A700026 : BOOL ;
    A700027 : BOOL ;
    A700028 : BOOL ;
    A700029 : BOOL ;
    A700030 : BOOL ;
    A700031 : BOOL ;
    A700032 : BOOL ;
    A700033 : BOOL ;
    A700034 : BOOL ;
    A700035 : BOOL ;
    A700036 : BOOL ;
    A700037 : BOOL ;
    A700038 : BOOL ;
    A700039 : BOOL ;
    A700040 : BOOL ;
    A700041 : BOOL ;
    A700042 : BOOL ;
    A700043 : BOOL ;
    A700044 : BOOL ;
    A700045 : BOOL ;
    A700046 : BOOL ;
    A700047 : BOOL ;
    A700048 : BOOL ;
    A700049 : BOOL ;
    A700050 : BOOL ;
    A700051 : BOOL ;
    A700052 : BOOL ;
    A700053 : BOOL ;
    A700054 : BOOL ;
    A700055 : BOOL ;
    A700056 : BOOL ;
    A700057 : BOOL ;
    A700058 : BOOL ;
    A700059 : BOOL ;
    A700060 : BOOL ;
    A700061 : BOOL ;
    A700062 : BOOL ;
    A700063 : BOOL ;
   END_STRUCT ;
  END_STRUCT ;	
BEGIN
END_DATA_BLOCK

DATA_BLOCK DB 4
AUTHOR : NUMERIK
FAMILY : _800D
NAME : Basics
VERSION : 1.5
  STRUCT
   BOfeld0 : WORD  := W#16#CD54;	//Channel 1-8 ever 18 Bits
   BOfeld2 : WORD  := W#16#3553;
   BOfeld4 : WORD  := W#16#D54C;
   BOfeld6 : WORD  := W#16#5533;
   BOfeld8 : WORD  := W#16#55CD;
   BOfeld10 : WORD  := W#16#5435;
   BOfeld12 : WORD  := W#16#53D5;
   BOfeld14 : WORD  := W#16#4C55;
   BOfeld16 : WORD  := W#16#3355;
   BOfeld18 : WORD  := W#16#5555;	//18 Axes/Spindles ever 2 Bit
   BOfeld20 : WORD  := W#16#5555;
   BOfeld22 : WORD  := W#16#F5F0;	//10 User data area ever 8 Bit (Begin: DBB23)
   BOfeld24 : WORD  := W#16#F0F0;
   BOfeld26 : WORD  := W#16#F0F0;
   BOfeld28 : WORD  := W#16#F0F0;
   BOfeld30 : WORD  := W#16#F0F0;
   BOfeld32 : WORD  := W#16#F0F0;
   BOfeld34 : WORD  := W#16#F0F0;
   BOfeld36 : WORD  := W#16#F0F0;
   BOfeld38 : WORD  := W#16#F0F0;
   BOfeld40 : WORD  := W#16#F0F0;
   BOfeld42 : WORD  := W#16#F0F0;
   BOfeld44 : WORD  := W#16#F0F0;
   BOfeld46 : WORD  := W#16#F0F0;
   BOfeld48 : WORD  := W#16#F0F0;
   BOfeld50 : WORD  := W#16#F0F0;
   BOfeld52 : WORD  := W#16#F0F0;
   BOfeld54 : WORD  := W#16#F0F0;
   BOfeld56 : WORD  := W#16#F0F0;
   BOfeld58 : WORD  := W#16#F0F0;
   BOfeld60 : WORD  := W#16#F0F0;
   BOfeld62 : BYTE  := B#16#F0;
   NumUser : BYTE  := B#16#A;
   maganz : BYTE ;	//for TM, number of Magazine
   wzv : BYTE ;
   wzvdat : ARRAY  [1 .. 160 ] OF BYTE ;	//32 Magazine, possibly ever 5 Byte + Spindle
  END_STRUCT ;	
BEGIN
   BOfeld0 := W#16#CD54;
   BOfeld2 := W#16#3553;
   BOfeld4 := W#16#D54C;
   BOfeld6 := W#16#5533;
   BOfeld8 := W#16#55CD;
   BOfeld10 := W#16#5435;
   BOfeld12 := W#16#53D5;
   BOfeld14 := W#16#4C55;
   BOfeld16 := W#16#3355;
   BOfeld18 := W#16#5555;
   BOfeld20 := W#16#5555;
   BOfeld22 := W#16#F5F0;
   BOfeld24 := W#16#F0F0;
   BOfeld26 := W#16#F0F0;
   BOfeld28 := W#16#F0F0;
   BOfeld30 := W#16#F0F0;
   BOfeld32 := W#16#F0F0;
   BOfeld34 := W#16#F0F0;
   BOfeld36 := W#16#F0F0;
   BOfeld38 := W#16#F0F0;
   BOfeld40 := W#16#F0F0;
   BOfeld42 := W#16#F0F0;
   BOfeld44 := W#16#F0F0;
   BOfeld46 := W#16#F0F0;
   BOfeld48 := W#16#F0F0;
   BOfeld50 := W#16#F0F0;
   BOfeld52 := W#16#F0F0;
   BOfeld54 := W#16#F0F0;
   BOfeld56 := W#16#F0F0;
   BOfeld58 := W#16#F0F0;
   BOfeld60 := W#16#F0F0;
   BOfeld62 := B#16#F0;
   NumUser := B#16#A;
END_DATA_BLOCK

